# B&R Automation Studio project Panasonic_LinkaPowerCP2_A2021055 (part 22)

#### AtlasCopcoKomunikacia.st
```iecst
ACTION AtlasCopcoKomunikacia:

    M5_PrevodMomentu();
    M4_PrevodMomentu();
    M6_PrevodMomentu();

	//*********************************************************Skrutkovacka M5******************************************************************//
	//Vstupy z AtlasCopco do PLC//
    P2_Srobovanie.Skrutkovacka_M5.Stav_VysledokPotvrdeny:= P2_Srobovanie.PAR.M5_AtlasCopcoInputs[0].0;
    P2_Srobovanie.Skrutkovacka_M5.Stav_EmergencyStop:= P2_Srobovanie.PAR.M5_AtlasCopcoInputs[0].1;
    P2_Srobovanie.Skrutkovacka_M5.Stav_READY_to_START:= P2_Srobovanie.PAR.M5_AtlasCopcoInputs[0].2;
    P2_Srobovanie.Skrutkovacka_M5.Stav_MANUAL:= P2_Srobovanie.PAR.M5_AtlasCopcoInputs[0].3;
    P2_Srobovanie.Skrutkovacka_M5.Stav_UtahovanieUkoncene:= P2_Srobovanie.PAR.M5_AtlasCopcoInputs[0].4;
    P2_Srobovanie.Skrutkovacka_M5.Stav_VysledokUtahovania_NG:= P2_Srobovanie.PAR.M5_AtlasCopcoInputs[0].5;
    P2_Srobovanie.Skrutkovacka_M5.Stav_VysledokUtahovania_OK:= P2_Srobovanie.PAR.M5_AtlasCopcoInputs[0].6;
    P2_Srobovanie.Skrutkovacka_M5.Stav_SmerOtacania_VPRED:= P2_Srobovanie.PAR.M5_AtlasCopcoInputs[0].7;
    P2_Srobovanie.Skrutkovacka_M5.Stav_BUSY:= P2_Srobovanie.PAR.M5_AtlasCopcoInputs[0].8;
    P2_Srobovanie.Skrutkovacka_M5.Stav_ControlerSwitch_ON:= P2_Srobovanie.PAR.M5_AtlasCopcoInputs[0].9;
    P2_Srobovanie.Skrutkovacka_M5.Stav_Station_READY:= P2_Srobovanie.PAR.M5_AtlasCopcoInputs[0].10;
    P2_Srobovanie.Skrutkovacka_M5.Stav_NastrojPripojeny:= P2_Srobovanie.PAR.M5_AtlasCopcoInputs[0].11;
    P2_Srobovanie.Skrutkovacka_M5.Stav_NastrojUtahuje:= P2_Srobovanie.PAR.M5_AtlasCopcoInputs[0].12;

    //Výstupy z PLC do AtlasCopco//
    P2_Srobovanie.PAR.M5_AtlasCopcoOutputs[0].0:= P2_Srobovanie.Skrutkovacka_M5.RESET_Poruchy;
    P2_Srobovanie.PAR.M5_AtlasCopcoOutputs[0].1:= P2_Srobovanie.Skrutkovacka_M5.RESET_Vysledkov;
    P2_Srobovanie.PAR.M5_AtlasCopcoOutputs[0].2:= P2_Srobovanie.Skrutkovacka_M5.START_Skrutkovania;
    P2_Srobovanie.PAR.M5_AtlasCopcoOutputs[0].3:= P2_Srobovanie.Skrutkovacka_M5.START_Utahovania;

    //Dosiahnutý moment//
//    P2_Srobovanie.STAV.M5_DosiahnutyMoment.0:= P2_Srobovanie.PAR.M5_AtlasCopcoInputs[1].24;
//    P2_Srobovanie.STAV.M5_DosiahnutyMoment.1:= P2_Srobovanie.PAR.M5_AtlasCopcoInputs[1].25;
//    P2_Srobovanie.STAV.M5_DosiahnutyMoment.2:= P2_Srobovanie.PAR.M5_AtlasCopcoInputs[1].26;
//    P2_Srobovanie.STAV.M5_DosiahnutyMoment.3:= P2_Srobovanie.PAR.M5_AtlasCopcoInputs[1].27;
//    P2_Srobovanie.STAV.M5_DosiahnutyMoment.4:= P2_Srobovanie.PAR.M5_AtlasCopcoInputs[1].28;
//    P2_Srobovanie.STAV.M5_DosiahnutyMoment.5:= P2_Srobovanie.PAR.M5_AtlasCopcoInputs[1].29;
//    P2_Srobovanie.STAV.M5_DosiahnutyMoment.6:= P2_Srobovanie.PAR.M5_AtlasCopcoInputs[1].30;
//    P2_Srobovanie.STAV.M5_DosiahnutyMoment.7:= P2_Srobovanie.PAR.M5_AtlasCopcoInputs[1].31;
//    P2_Srobovanie.STAV.M5_DosiahnutyMoment.8:= P2_Srobovanie.PAR.M5_AtlasCopcoInputs[1].16;
//    P2_Srobovanie.STAV.M5_DosiahnutyMoment.9:= P2_Srobovanie.PAR.M5_AtlasCopcoInputs[1].17;
//    P2_Srobovanie.STAV.M5_DosiahnutyMoment.10:= P2_Srobovanie.PAR.M5_AtlasCopcoInputs[1].18;
//    P2_Srobovanie.STAV.M5_DosiahnutyMoment.11:= P2_Srobovanie.PAR.M5_AtlasCopcoInputs[1].19;
//    P2_Srobovanie.STAV.M5_DosiahnutyMoment.12:= P2_Srobovanie.PAR.M5_AtlasCopcoInputs[1].20;
//    P2_Srobovanie.STAV.M5_DosiahnutyMoment.13:= P2_Srobovanie.PAR.M5_AtlasCopcoInputs[1].21;
//    P2_Srobovanie.STAV.M5_DosiahnutyMoment.14:= P2_Srobovanie.PAR.M5_AtlasCopcoInputs[1].22;
//    P2_Srobovanie.STAV.M5_DosiahnutyMoment.15:= P2_Srobovanie.PAR.M5_AtlasCopcoInputs[1].23;
//    P2_Srobovanie.STAV.M5_DosiahnutyMoment.16:= P2_Srobovanie.PAR.M5_AtlasCopcoInputs[1].8;
//    P2_Srobovanie.STAV.M5_DosiahnutyMoment.17:= P2_Srobovanie.PAR.M5_AtlasCopcoInputs[1].9;
//    P2_Srobovanie.STAV.M5_DosiahnutyMoment.18:= P2_Srobovanie.PAR.M5_AtlasCopcoInputs[1].10;
//    P2_Srobovanie.STAV.M5_DosiahnutyMoment.19:= P2_Srobovanie.PAR.M5_AtlasCopcoInputs[1].11;
//    P2_Srobovanie.STAV.M5_DosiahnutyMoment.20:= P2_Srobovanie.PAR.M5_AtlasCopcoInputs[1].12;
//    P2_Srobovanie.STAV.M5_DosiahnutyMoment.21:= P2_Srobovanie.PAR.M5_AtlasCopcoInputs[1].13;
//    P2_Srobovanie.STAV.M5_DosiahnutyMoment.22:= P2_Srobovanie.PAR.M5_AtlasCopcoInputs[1].14;
//    P2_Srobovanie.STAV.M5_DosiahnutyMoment.23:= P2_Srobovanie.PAR.M5_AtlasCopcoInputs[1].15;
//    P2_Srobovanie.STAV.M5_DosiahnutyMoment.24:= P2_Srobovanie.PAR.M5_AtlasCopcoInputs[1].0;
//    P2_Srobovanie.STAV.M5_DosiahnutyMoment.25:= P2_Srobovanie.PAR.M5_AtlasCopcoInputs[1].1;
//    P2_Srobovanie.STAV.M5_DosiahnutyMoment.26:= P2_Srobovanie.PAR.M5_AtlasCopcoInputs[1].2;
//    P2_Srobovanie.STAV.M5_DosiahnutyMoment.27:= P2_Srobovanie.PAR.M5_AtlasCopcoInputs[1].3;
//    P2_Srobovanie.STAV.M5_DosiahnutyMoment.28:= P2_Srobovanie.PAR.M5_AtlasCopcoInputs[1].4;
//    P2_Srobovanie.STAV.M5_DosiahnutyMoment.29:= P2_Srobovanie.PAR.M5_AtlasCopcoInputs[1].5;
//    P2_Srobovanie.STAV.M5_DosiahnutyMoment.30:= P2_Srobovanie.PAR.M5_AtlasCopcoInputs[1].6;
//    P2_Srobovanie.STAV.M5_DosiahnutyMoment.31:= P2_Srobovanie.PAR.M5_AtlasCopcoInputs[1].7;
//    M5_DosiahnutyMoment_REAL:= UDINT_TO_REAL(P2_Srobovanie.STAV.M5_DosiahnutyMoment);
//    IF M5_DosiahnutyMoment_REAL > 0 THEN
//        P2_Srobovanie.STAV.M5_DosiahnutyMoment_REAL:= M5_DosiahnutyMoment_REAL/100;
//    ELSE
//        P2_Srobovanie.STAV.M5_DosiahnutyMoment_REAL:= 0.0;
//    END_IF

    M5_PrevodMomentu.AtlasAktualnyMoment:=P2_Srobovanie.PAR.M5_AtlasCopcoInputs[1];
    P2_Srobovanie.STAV.M5_DosiahnutyMoment_REAL:=M5_PrevodMomentu.AktualnyMoment;

    //Moment - Tolerancia MAX//
//    P2_Srobovanie.STAV.M5_Moment_ToleranciaMAX.0:= P2_Srobovanie.PAR.M5_AtlasCopcoInputs[3].24;
//    P2_Srobovanie.STAV.M5_Moment_ToleranciaMAX.1:= P2_Srobovanie.PAR.M5_AtlasCopcoInputs[3].25;
//    P2_Srobovanie.STAV.M5_Moment_ToleranciaMAX.2:= P2_Srobovanie.PAR.M5_AtlasCopcoInputs[3].26;
//    P2_Srobovanie.STAV.M5_Moment_ToleranciaMAX.3:= P2_Srobovanie.PAR.M5_AtlasCopcoInputs[3].27;
//    P2_Srobovanie.STAV.M5_Moment_ToleranciaMAX.4:= P2_Srobovanie.PAR.M5_AtlasCopcoInputs[3].28;
//    P2_Srobovanie.STAV.M5_Moment_ToleranciaMAX.5:= P2_Srobovanie.PAR.M5_AtlasCopcoInputs[3].29;
//    P2_Srobovanie.STAV.M5_Moment_ToleranciaMAX.6:= P2_Srobovanie.PAR.M5_AtlasCopcoInputs[3].30;
//    P2_Srobovanie.STAV.M5_Moment_ToleranciaMAX.7:= P2_Srobovanie.PAR.M5_AtlasCopcoInputs[3].31;
//    P2_Srobovanie.STAV.M5_Moment_ToleranciaMAX.8:= P2_Srobovanie.PAR.M5_AtlasCopcoInputs[3].16;
//    P2_Srobovanie.STAV.M5_Moment_ToleranciaMAX.9:= P2_Srobovanie.PAR.M5_AtlasCopcoInputs[3].17;
//    P2_Srobovanie.STAV.M5_Moment_ToleranciaMAX.10:= P2_Srobovanie.PAR.M5_AtlasCopcoInputs[3].18;
//    P2_Srobovanie.STAV.M5_Moment_ToleranciaMAX.11:= P2_Srobovanie.PAR.M5_AtlasCopcoInputs[3].19;
//    P2_Srobovanie.STAV.M5_Moment_ToleranciaMAX.12:= P2_Srobovanie.PAR.M5_AtlasCopcoInputs[3].20;
//    P2_Srobovanie.STAV.M5_Moment_ToleranciaMAX.13:= P2_Srobovanie.PAR.M5_AtlasCopcoInputs[3].21;
//    P2_Srobovanie.STAV.M5_Moment_ToleranciaMAX.14:= P2_Srobovanie.PAR.M5_AtlasCopcoInputs[3].22;
//    P2_Srobovanie.STAV.M5_Moment_ToleranciaMAX.15:= P2_Srobovanie.PAR.M5_AtlasCopcoInputs[3].23;
//    P2_Srobovanie.STAV.M5_Moment_ToleranciaMAX.16:= P2_Srobovanie.PAR.M5_AtlasCopcoInputs[3].8;
//    P2_Srobovanie.STAV.M5_Moment_ToleranciaMAX.17:= P2_Srobovanie.PAR.M5_AtlasCopcoInputs[3].9;
//    P2_Srobovanie.STAV.M5_Moment_ToleranciaMAX.18:= P2_Srobovanie.PAR.M5_AtlasCopcoInputs[3].10;
//    P2_Srobovanie.STAV.M5_Moment_ToleranciaMAX.19:= P2_Srobovanie.PAR.M5_AtlasCopcoInputs[3].11;
//    P2_Srobovanie.STAV.M5_Moment_ToleranciaMAX.20:= P2_Srobovanie.PAR.M5_AtlasCopcoInputs[3].12;
//    P2_Srobovanie.STAV.M5_Moment_ToleranciaMAX.21:= P2_Srobovanie.PAR.M5_AtlasCopcoInputs[3].13;
//    P2_Srobovanie.STAV.M5_Moment_ToleranciaMAX.22:= P2_Srobovanie.PAR.M5_AtlasCopcoInputs[3].14;
//    P2_Srobovanie.STAV.M5_Moment_ToleranciaMAX.23:= P2_Srobovanie.PAR.M5_AtlasCopcoInputs[3].15;
//    P2_Srobovanie.STAV.M5_Moment_ToleranciaMAX.24:= P2_Srobovanie.PAR.M5_AtlasCopcoInputs[3].0;
//    P2_Srobovanie.STAV.M5_Moment_ToleranciaMAX.25:= P2_Srobovanie.PAR.M5_AtlasCopcoInputs[3].1;
//    P2_Srobovanie.STAV.M5_Moment_ToleranciaMAX.26:= P2_Srobovanie.PAR.M5_AtlasCopcoInputs[3].2;
//    P2_Srobovanie.STAV.M5_Moment_ToleranciaMAX.27:= P2_Srobovanie.PAR.M5_AtlasCopcoInputs[3].3;
//    P2_Srobovanie.STAV.M5_Moment_ToleranciaMAX.28:= P2_Srobovanie.PAR.M5_AtlasCopcoInputs[3].4;
//    P2_Srobovanie.STAV.M5_Moment_ToleranciaMAX.29:= P2_Srobovanie.PAR.M5_AtlasCopcoInputs[3].5;
//    P2_Srobovanie.STAV.M5_Moment_ToleranciaMAX.30:= P2_Srobovanie.PAR.M5_AtlasCopcoInputs[3].6;
//    P2_Srobovanie.STAV.M5_Moment_ToleranciaMAX.31:= P2_Srobovanie.PAR.M5_AtlasCopcoInputs[3].7;
//    M5_Moment_ToleranciaMAX_REAL:= UDINT_TO_REAL(P2_Srobovanie.STAV.M5_Moment_ToleranciaMAX);
//    IF M5_Moment_ToleranciaMAX_REAL > 0 THEN
//        P2_Srobovanie.STAV.M5_Moment_ToleranciaMAX_REAL:= M5_Moment_ToleranciaMAX_REAL/100;
//    ELSE
//        P2_Srobovanie.STAV.M5_Moment_ToleranciaMAX_REAL:= 0.0;
//    END_IF

    M5_PrevodMomentu.AtlasMaximalnaTolerancia:=P2_Srobovanie.PAR.M5_AtlasCopcoInputs[3];
    P2_Srobovanie.STAV.M5_Moment_ToleranciaMAX_REAL:=M5_PrevodMomentu.ToleranciaMAX;

    //Moment - Tolerancia MIN//
//    P2_Srobovanie.STAV.M5_Moment_ToleranciaMIN.0:= P2_Srobovanie.PAR.M5_AtlasCopcoInputs[4].24;
//    P2_Srobovanie.STAV.M5_Moment_ToleranciaMIN.1:= P2_Srobovanie.PAR.M5_AtlasCopcoInputs[4].25;
//    P2_Srobovanie.STAV.M5_Moment_ToleranciaMIN.2:= P2_Srobovanie.PAR.M5_AtlasCopcoInputs[4].26;
//    P2_Srobovanie.STAV.M5_Moment_ToleranciaMIN.3:= P2_Srobovanie.PAR.M5_AtlasCopcoInputs[4].27;
//    P2_Srobovanie.STAV.M5_Moment_ToleranciaMIN.4:= P2_Srobovanie.PAR.M5_AtlasCopcoInputs[4].28;
//    P2_Srobovanie.STAV.M5_Moment_ToleranciaMIN.5:= P2_Srobovanie.PAR.M5_AtlasCopcoInputs[4].29;
//    P2_Srobovanie.STAV.M5_Moment_ToleranciaMIN.6:= P2_Srobovanie.PAR.M5_AtlasCopcoInputs[4].30;
//    P2_Srobovanie.STAV.M5_Moment_ToleranciaMIN.7:= P2_Srobovanie.PAR.M5_AtlasCopcoInputs[4].31;
//    P2_Srobovanie.STAV.M5_Moment_ToleranciaMIN.8:= P2_Srobovanie.PAR.M5_AtlasCopcoInputs[4].16;
//    P2_Srobovanie.STAV.M5_Moment_ToleranciaMIN.9:= P2_Srobovanie.PAR.M5_AtlasCopcoInputs[4].17;
//    P2_Srobovanie.STAV.M5_Moment_ToleranciaMIN.10:= P2_Srobovanie.PAR.M5_AtlasCopcoInputs[4].18;
//    P2_Srobovanie.STAV.M5_Moment_ToleranciaMIN.11:= P2_Srobovanie.PAR.M5_AtlasCopcoInputs[4].19;
//    P2_Srobovanie.STAV.M5_Moment_ToleranciaMIN.12:= P2_Srobovanie.PAR.M5_AtlasCopcoInputs[4].20;
//    P2_Srobovanie.STAV.M5_Moment_ToleranciaMIN.13:= P2_Srobovanie.PAR.M5_AtlasCopcoInputs[4].21;
//    P2_Srobovanie.STAV.M5_Moment_ToleranciaMIN.14:= P2_Srobovanie.PAR.M5_AtlasCopcoInputs[4].22;
//    P2_Srobovanie.STAV.M5_Moment_ToleranciaMIN.15:= P2_Srobovanie.PAR.M5_AtlasCopcoInputs[4].23;
//    P2_Srobovanie.STAV.M5_Moment_ToleranciaMIN.16:= P2_Srobovanie.PAR.M5_AtlasCopcoInputs[4].8;
//    P2_Srobovanie.STAV.M5_Moment_ToleranciaMIN.17:= P2_Srobovanie.PAR.M5_AtlasCopcoInputs[4].9;
//    P2_Srobovanie.STAV.M5_Moment_ToleranciaMIN.18:= P2_Srobovanie.PAR.M5_AtlasCopcoInputs[4].10;
//    P2_Srobovanie.STAV.M5_Moment_ToleranciaMIN.19:= P2_Srobovanie.PAR.M5_AtlasCopcoInputs[4].11;
//    P2_Srobovanie.STAV.M5_Moment_ToleranciaMIN.20:= P2_Srobovanie.PAR.M5_AtlasCopcoInputs[4].12;
//    P2_Srobovanie.STAV.M5_Moment_ToleranciaMIN.21:= P2_Srobovanie.PAR.M5_AtlasCopcoInputs[4].13;
//    P2_Srobovanie.STAV.M5_Moment_ToleranciaMIN.22:= P2_Srobovanie.PAR.M5_AtlasCopcoInputs[4].14;
//    P2_Srobovanie.STAV.M5_Moment_ToleranciaMIN.23:= P2_Srobovanie.PAR.M5_AtlasCopcoInputs[4].15;
//    P2_Srobovanie.STAV.M5_Moment_ToleranciaMIN.24:= P2_Srobovanie.PAR.M5_AtlasCopcoInputs[4].0;
//    P2_Srobovanie.STAV.M5_Moment_ToleranciaMIN.25:= P2_Srobovanie.PAR.M5_AtlasCopcoInputs[4].1;
//    P2_Srobovanie.STAV.M5_Moment_ToleranciaMIN.26:= P2_Srobovanie.PAR.M5_AtlasCopcoInputs[4].2;
//    P2_Srobovanie.STAV.M5_Moment_ToleranciaMIN.27:= P2_Srobovanie.PAR.M5_AtlasCopcoInputs[4].3;
//    P2_Srobovanie.STAV.M5_Moment_ToleranciaMIN.28:= P2_Srobovanie.PAR.M5_AtlasCopcoInputs[4].4;
//    P2_Srobovanie.STAV.M5_Moment_ToleranciaMIN.29:= P2_Srobovanie.PAR.M5_AtlasCopcoInputs[4].5;
//    P2_Srobovanie.STAV.M5_Moment_ToleranciaMIN.30:= P2_Srobovanie.PAR.M5_AtlasCopcoInputs[4].6;
//    P2_Srobovanie.STAV.M5_Moment_ToleranciaMIN.31:= P2_Srobovanie.PAR.M5_AtlasCopcoInputs[4].7;
//    M5_Moment_ToleranciaMIN_REAL:= UDINT_TO_REAL(P2_Srobovanie.STAV.M5_Moment_ToleranciaMIN);
//    IF M5_Moment_ToleranciaMIN_REAL > 0 THEN
//        P2_Srobovanie.STAV.M5_Moment_ToleranciaMIN_REAL:= M5_Moment_ToleranciaMIN_REAL /100;
//    ELSE
//        P2_Srobovanie.STAV.M5_Moment_ToleranciaMIN_REAL:= 0.0;
    //    END_IF

    M5_PrevodMomentu.AtlasMinimalnaTolerancia:=P2_Srobovanie.PAR.M5_AtlasCopcoInputs[4];
    P2_Srobovanie.STAV.M5_Moment_ToleranciaMIN_REAL:=M5_PrevodMomentu.ToleranciaMIN;

    //Dosiahnutý úhol//
    P2_Srobovanie.STAV.M5_DosiahnutyUhol.0:= P2_Srobovanie.PAR.M5_AtlasCopcoInputs[0].24;
    P2_Srobovanie.STAV.M5_DosiahnutyUhol.1:= P2_Srobovanie.PAR.M5_AtlasCopcoInputs[0].25;
    P2_Srobovanie.STAV.M5_DosiahnutyUhol.2:= P2_Srobovanie.PAR.M5_AtlasCopcoInputs[0].26;
    P2_Srobovanie.STAV.M5_DosiahnutyUhol.3:= P2_Srobovanie.PAR.M5_AtlasCopcoInputs[0].27;
    P2_Srobovanie.STAV.M5_DosiahnutyUhol.4:= P2_Srobovanie.PAR.M5_AtlasCopcoInputs[0].28;
    P2_Srobovanie.STAV.M5_DosiahnutyUhol.5:= P2_Srobovanie.PAR.M5_AtlasCopcoInputs[0].29;
    P2_Srobovanie.STAV.M5_DosiahnutyUhol.6:= P2_Srobovanie.PAR.M5_AtlasCopcoInputs[0].30;
    P2_Srobovanie.STAV.M5_DosiahnutyUhol.7:= P2_Srobovanie.PAR.M5_AtlasCopcoInputs[0].31;
    P2_Srobovanie.STAV.M5_DosiahnutyUhol.8:= P2_Srobovanie.PAR.M5_AtlasCopcoInputs[0].16;
    P2_Srobovanie.STAV.M5_DosiahnutyUhol.9:= P2_Srobovanie.PAR.M5_AtlasCopcoInputs[0].17;
    P2_Srobovanie.STAV.M5_DosiahnutyUhol.10:= P2_Srobovanie.PAR.M5_AtlasCopcoInputs[0].18;
    P2_Srobovanie.STAV.M5_DosiahnutyUhol.11:= P2_Srobovanie.PAR.M5_AtlasCopcoInputs[0].19;
    P2_Srobovanie.STAV.M5_DosiahnutyUhol.12:= P2_Srobovanie.PAR.M5_AtlasCopcoInputs[0].20;
    P2_Srobovanie.STAV.M5_DosiahnutyUhol.13:= P2_Srobovanie.PAR.M5_AtlasCopcoInputs[0].21;
    P2_Srobovanie.STAV.M5_DosiahnutyUhol.14:= P2_Srobovanie.PAR.M5_AtlasCopcoInputs[0].22;
    P2_Srobovanie.STAV.M5_DosiahnutyUhol.15:= P2_Srobovanie.PAR.M5_AtlasCopcoInputs[0].23;

    //Uhol - Tolerancia MAX//
    P2_Srobovanie.STAV.M5_Uhol_ToleranciaMAX.0:= P2_Srobovanie.PAR.M5_AtlasCopcoInputs[2].8;
    P2_Srobovanie.STAV.M5_Uhol_ToleranciaMAX.1:= P2_Srobovanie.PAR.M5_AtlasCopcoInputs[2].9;
    P2_Srobovanie.STAV.M5_Uhol_ToleranciaMAX.2:= P2_Srobovanie.PAR.M5_AtlasCopcoInputs[2].10;
    P2_Srobovanie.STAV.M5_Uhol_ToleranciaMAX.3:= P2_Srobovanie.PAR.M5_AtlasCopcoInputs[2].11;
    P2_Srobovanie.STAV.M5_Uhol_ToleranciaMAX.4:= P2_Srobovanie.PAR.M5_AtlasCopcoInputs[2].12;
    P2_Srobovanie.STAV.M5_Uhol_ToleranciaMAX.5:= P2_Srobovanie.PAR.M5_AtlasCopcoInputs[2].13;
    P2_Srobovanie.STAV.M5_Uhol_ToleranciaMAX.6:= P2_Srobovanie.PAR.M5_AtlasCopcoInputs[2].14;
    P2_Srobovanie.STAV.M5_Uhol_ToleranciaMAX.7:= P2_Srobovanie.PAR.M5_AtlasCopcoInputs[2].15;
    P2_Srobovanie.STAV.M5_Uhol_ToleranciaMAX.8:= P2_Srobovanie.PAR.M5_AtlasCopcoInputs[2].0;
    P2_Srobovanie.STAV.M5_Uhol_ToleranciaMAX.9:= P2_Srobovanie.PAR.M5_AtlasCopcoInputs[2].1;
    P2_Srobovanie.STAV.M5_Uhol_ToleranciaMAX.10:= P2_Srobovanie.PAR.M5_AtlasCopcoInputs[2].2;
    P2_Srobovanie.STAV.M5_Uhol_ToleranciaMAX.11:= P2_Srobovanie.PAR.M5_AtlasCopcoInputs[2].3;
    P2_Srobovanie.STAV.M5_Uhol_ToleranciaMAX.12:= P2_Srobovanie.PAR.M5_AtlasCopcoInputs[2].4;
    P2_Srobovanie.STAV.M5_Uhol_ToleranciaMAX.13:= P2_Srobovanie.PAR.M5_AtlasCopcoInputs[2].5;
    P2_Srobovanie.STAV.M5_Uhol_ToleranciaMAX.14:= P2_Srobovanie.PAR.M5_AtlasCopcoInputs[2].6;
    P2_Srobovanie.STAV.M5_Uhol_ToleranciaMAX.15:= P2_Srobovanie.PAR.M5_AtlasCopcoInputs[2].7;

    //Uhol - Tolerancia MIN//
    P2_Srobovanie.STAV.M5_Uhol_ToleranciaMIN.0:= P2_Srobovanie.PAR.M5_AtlasCopcoInputs[2].24;
    P2_Srobovanie.STAV.M5_Uhol_ToleranciaMIN.1:= P2_Srobovanie.PAR.M5_AtlasCopcoInputs[2].25;
    P2_Srobovanie.STAV.M5_Uhol_ToleranciaMIN.2:= P2_Srobovanie.PAR.M5_AtlasCopcoInputs[2].26;
    P2_Srobovanie.STAV.M5_Uhol_ToleranciaMIN.3:= P2_Srobovanie.PAR.M5_AtlasCopcoInputs[2].27;
    P2_Srobovanie.STAV.M5_Uhol_ToleranciaMIN.4:= P2_Srobovanie.PAR.M5_AtlasCopcoInputs[2].28;
    P2_Srobovanie.STAV.M5_Uhol_ToleranciaMIN.5:= P2_Srobovanie.PAR.M5_AtlasCopcoInputs[2].29;
    P2_Srobovanie.STAV.M5_Uhol_ToleranciaMIN.6:= P2_Srobovanie.PAR.M5_AtlasCopcoInputs[2].30;
    P2_Srobovanie.STAV.M5_Uhol_ToleranciaMIN.7:= P2_Srobovanie.PAR.M5_AtlasCopcoInputs[2].31;
    P2_Srobovanie.STAV.M5_Uhol_ToleranciaMIN.8:= P2_Srobovanie.PAR.M5_AtlasCopcoInputs[2].16;
    P2_Srobovanie.STAV.M5_Uhol_ToleranciaMIN.9:= P2_Srobovanie.PAR.M5_AtlasCopcoInputs[2].17;
    P2_Srobovanie.STAV.M5_Uhol_ToleranciaMIN.10:= P2_Srobovanie.PAR.M5_AtlasCopcoInputs[2].18;
    P2_Srobovanie.STAV.M5_Uhol_ToleranciaMIN.11:= P2_Srobovanie.PAR.M5_AtlasCopcoInputs[2].19;
    P2_Srobovanie.STAV.M5_Uhol_ToleranciaMIN.12:= P2_Srobovanie.PAR.M5_AtlasCopcoInputs[2].20;
    P2_Srobovanie.STAV.M5_Uhol_ToleranciaMIN.13:= P2_Srobovanie.PAR.M5_AtlasCopcoInputs[2].21;
    P2_Srobovanie.STAV.M5_Uhol_ToleranciaMIN.14:= P2_Srobovanie.PAR.M5_AtlasCopcoInputs[2].22;
    P2_Srobovanie.STAV.M5_Uhol_ToleranciaMIN.15:= P2_Srobovanie.PAR.M5_AtlasCopcoInputs[2].23;

    //*****************************************************************************Skrutkovacka M4*************************************************************//
    //Vstupy z AtlasCopco do PLC//
    P2_Srobovanie.Skrutkovacka_M4.Stav_VysledokPotvrdeny:= P2_Srobovanie.PAR.M4_AtlasCopcoInputs[0].0;
    P2_Srobovanie.Skrutkovacka_M4.Stav_EmergencyStop:= P2_Srobovanie.PAR.M4_AtlasCopcoInputs[0].1;
    P2_Srobovanie.Skrutkovacka_M4.Stav_READY_to_START:= P2_Srobovanie.PAR.M4_AtlasCopcoInputs[0].2;
    P2_Srobovanie.Skrutkovacka_M4.Stav_MANUAL:= P2_Srobovanie.PAR.M4_AtlasCopcoInputs[0].3;
    P2_Srobovanie.Skrutkovacka_M4.Stav_UtahovanieUkoncene:= P2_Srobovanie.PAR.M4_AtlasCopcoInputs[0].4;
    P2_Srobovanie.Skrutkovacka_M4.Stav_VysledokUtahovania_NG:= P2_Srobovanie.PAR.M4_AtlasCopcoInputs[0].5;
    P2_Srobovanie.Skrutkovacka_M4.Stav_VysledokUtahovania_OK:= P2_Srobovanie.PAR.M4_AtlasCopcoInputs[0].6;
    P2_Srobovanie.Skrutkovacka_M4.Stav_SmerOtacania_VPRED:= P2_Srobovanie.PAR.M4_AtlasCopcoInputs[0].7;
    P2_Srobovanie.Skrutkovacka_M4.Stav_BUSY:= P2_Srobovanie.PAR.M4_AtlasCopcoInputs[0].8;
    P2_Srobovanie.Skrutkovacka_M4.Stav_ControlerSwitch_ON:= P2_Srobovanie.PAR.M4_AtlasCopcoInputs[0].9;
    P2_Srobovanie.Skrutkovacka_M4.Stav_Station_READY:= P2_Srobovanie.PAR.M4_AtlasCopcoInputs[0].10;
    P2_Srobovanie.Skrutkovacka_M4.Stav_NastrojPripojeny:= P2_Srobovanie.PAR.M4_AtlasCopcoInputs[0].11;
    P2_Srobovanie.Skrutkovacka_M4.Stav_NastrojUtahuje:= P2_Srobovanie.PAR.M4_AtlasCopcoInputs[0].12;

    //Výstupy z PLC do AtlasCopco//
    P2_Srobovanie.PAR.M4_AtlasCopcoOutputs[0].0:= P2_Srobovanie.Skrutkovacka_M4.RESET_Poruchy;
    P2_Srobovanie.PAR.M4_AtlasCopcoOutputs[0].1:= P2_Srobovanie.Skrutkovacka_M4.RESET_Vysledkov;
    P2_Srobovanie.PAR.M4_AtlasCopcoOutputs[0].2:= P2_Srobovanie.Skrutkovacka_M4.START_Skrutkovania;
    P2_Srobovanie.PAR.M4_AtlasCopcoOutputs[0].3:= P2_Srobovanie.Skrutkovacka_M4.START_Utahovania;

    //Dosiahnutý moment//
//    P2_Srobovanie.STAV.M4_DosiahnutyMoment.0:= P2_Srobovanie.PAR.M4_AtlasCopcoInputs[1].24;
//    P2_Srobovanie.STAV.M4_DosiahnutyMoment.1:= P2_Srobovanie.PAR.M4_AtlasCopcoInputs[1].25;
//    P2_Srobovanie.STAV.M4_DosiahnutyMoment.2:= P2_Srobovanie.PAR.M4_AtlasCopcoInputs[1].26;
//    P2_Srobovanie.STAV.M4_DosiahnutyMoment.3:= P2_Srobovanie.PAR.M4_AtlasCopcoInputs[1].27;
//    P2_Srobovanie.STAV.M4_DosiahnutyMoment.4:= P2_Srobovanie.PAR.M4_AtlasCopcoInputs[1].28;
//    P2_Srobovanie.STAV.M4_DosiahnutyMoment.5:= P2_Srobovanie.PAR.M4_AtlasCopcoInputs[1].29;
//    P2_Srobovanie.STAV.M4_DosiahnutyMoment.6:= P2_Srobovanie.PAR.M4_AtlasCopcoInputs[1].30;
//    P2_Srobovanie.STAV.M4_DosiahnutyMoment.7:= P2_Srobovanie.PAR.M4_AtlasCopcoInputs[1].31;
//    P2_Srobovanie.STAV.M4_DosiahnutyMoment.8:= P2_Srobovanie.PAR.M4_AtlasCopcoInputs[1].16;
//    P2_Srobovanie.STAV.M4_DosiahnutyMoment.9:= P2_Srobovanie.PAR.M4_AtlasCopcoInputs[1].17;
//    P2_Srobovanie.STAV.M4_DosiahnutyMoment.10:= P2_Srobovanie.PAR.M4_AtlasCopcoInputs[1].18;
//    P2_Srobovanie.STAV.M4_DosiahnutyMoment.11:= P2_Srobovanie.PAR.M4_AtlasCopcoInputs[1].19;
//    P2_Srobovanie.STAV.M4_DosiahnutyMoment.12:= P2_Srobovanie.PAR.M4_AtlasCopcoInputs[1].20;
//    P2_Srobovanie.STAV.M4_DosiahnutyMoment.13:= P2_Srobovanie.PAR.M4_AtlasCopcoInputs[1].21;
//    P2_Srobovanie.STAV.M4_DosiahnutyMoment.14:= P2_Srobovanie.PAR.M4_AtlasCopcoInputs[1].22;
//    P2_Srobovanie.STAV.M4_DosiahnutyMoment.15:= P2_Srobovanie.PAR.M4_AtlasCopcoInputs[1].23;
//    P2_Srobovanie.STAV.M4_DosiahnutyMoment.16:= P2_Srobovanie.PAR.M4_AtlasCopcoInputs[1].8;
//    P2_Srobovanie.STAV.M4_DosiahnutyMoment.17:= P2_Srobovanie.PAR.M4_AtlasCopcoInputs[1].9;
//    P2_Srobovanie.STAV.M4_DosiahnutyMoment.18:= P2_Srobovanie.PAR.M4_AtlasCopcoInputs[1].10;
//    P2_Srobovanie.STAV.M4_DosiahnutyMoment.19:= P2_Srobovanie.PAR.M4_AtlasCopcoInputs[1].11;
//    P2_Srobovanie.STAV.M4_DosiahnutyMoment.20:= P2_Srobovanie.PAR.M4_AtlasCopcoInputs[1].12;
//    P2_Srobovanie.STAV.M4_DosiahnutyMoment.21:= P2_Srobovanie.PAR.M4_AtlasCopcoInputs[1].13;
//    P2_Srobovanie.STAV.M4_DosiahnutyMoment.22:= P2_Srobovanie.PAR.M4_AtlasCopcoInputs[1].14;
//    P2_Srobovanie.STAV.M4_DosiahnutyMoment.23:= P2_Srobovanie.PAR.M4_AtlasCopcoInputs[1].15;
//    P2_Srobovanie.STAV.M4_DosiahnutyMoment.24:= P2_Srobovanie.PAR.M4_AtlasCopcoInputs[1].0;
//    P2_Srobovanie.STAV.M4_DosiahnutyMoment.25:= P2_Srobovanie.PAR.M4_AtlasCopcoInputs[1].1;
//    P2_Srobovanie.STAV.M4_DosiahnutyMoment.26:= P2_Srobovanie.PAR.M4_AtlasCopcoInputs[1].2;
//    P2_Srobovanie.STAV.M4_DosiahnutyMoment.27:= P2_Srobovanie.PAR.M4_AtlasCopcoInputs[1].3;
//    P2_Srobovanie.STAV.M4_DosiahnutyMoment.28:= P2_Srobovanie.PAR.M4_AtlasCopcoInputs[1].4;
//    P2_Srobovanie.STAV.M4_DosiahnutyMoment.29:= P2_Srobovanie.PAR.M4_AtlasCopcoInputs[1].5;
//    P2_Srobovanie.STAV.M4_DosiahnutyMoment.30:= P2_Srobovanie.PAR.M4_AtlasCopcoInputs[1].6;
//    P2_Srobovanie.STAV.M4_DosiahnutyMoment.31:= P2_Srobovanie.PAR.M4_AtlasCopcoInputs[1].7;
//    M4_DosiahnutyMoment_REAL:= UDINT_TO_REAL(P2_Srobovanie.STAV.M4_DosiahnutyMoment);
//    IF M4_DosiahnutyMoment_REAL > 0 THEN
//      P2_Srobovanie.STAV.M4_DosiahnutyMoment_REAL:= (M4_DosiahnutyMoment_REAL*2.1)/131082;
//    ELSE
//        P2_Srobovanie.STAV.M4_DosiahnutyMoment_REAL:= 0.0;
//    END_IF
//    (*P2_Srobovanie.STAV.M4_DosiahnutyMoment_REAL:= M4_DosiahnutyMoment_REAL/100;*)

    M4_PrevodMomentu.AtlasAktualnyMoment:=P2_Srobovanie.PAR.M4_AtlasCopcoInputs[1];
    P2_Srobovanie.STAV.M4_DosiahnutyMoment_REAL:=M4_PrevodMomentu.AktualnyMoment;

    //Moment - Tolerancia MAX//
//    P2_Srobovanie.STAV.M4_Moment_ToleranciaMAX.0:= P2_Srobovanie.PAR.M4_AtlasCopcoInputs[3].24;
//    P2_Srobovanie.STAV.M4_Moment_ToleranciaMAX.1:= P2_Srobovanie.PAR.M4_AtlasCopcoInputs[3].25;
//    P2_Srobovanie.STAV.M4_Moment_ToleranciaMAX.2:= P2_Srobovanie.PAR.M4_AtlasCopcoInputs[3].26;
//    P2_Srobovanie.STAV.M4_Moment_ToleranciaMAX.3:= P2_Srobovanie.PAR.M4_AtlasCopcoInputs[3].27;
//    P2_Srobovanie.STAV.M4_Moment_ToleranciaMAX.4:= P2_Srobovanie.PAR.M4_AtlasCopcoInputs[3].28;
//    P2_Srobovanie.STAV.M4_Moment_ToleranciaMAX.5:= P2_Srobovanie.PAR.M4_AtlasCopcoInputs[3].29;
//    P2_Srobovanie.STAV.M4_Moment_ToleranciaMAX.6:= P2_Srobovanie.PAR.M4_AtlasCopcoInputs[3].30;
//    P2_Srobovanie.STAV.M4_Moment_ToleranciaMAX.7:= P2_Srobovanie.PAR.M4_AtlasCopcoInputs[3].31;
//    P2_Srobovanie.STAV.M4_Moment_ToleranciaMAX.8:= P2_Srobovanie.PAR.M4_AtlasCopcoInputs[3].16;
//    P2_Srobovanie.STAV.M4_Moment_ToleranciaMAX.9:= P2_Srobovanie.PAR.M4_AtlasCopcoInputs[3].17;
//    P2_Srobovanie.STAV.M4_Moment_ToleranciaMAX.10:= P2_Srobovanie.PAR.M4_AtlasCopcoInputs[3].18;
//    P2_Srobovanie.STAV.M4_Moment_ToleranciaMAX.11:= P2_Srobovanie.PAR.M4_AtlasCopcoInputs[3].19;
//    P2_Srobovanie.STAV.M4_Moment_ToleranciaMAX.12:= P2_Srobovanie.PAR.M4_AtlasCopcoInputs[3].20;
//    P2_Srobovanie.STAV.M4_Moment_ToleranciaMAX.13:= P2_Srobovanie.PAR.M4_AtlasCopcoInputs[3].21;
//    P2_Srobovanie.STAV.M4_Moment_ToleranciaMAX.14:= P2_Srobovanie.PAR.M4_AtlasCopcoInputs[3].22;
//    P2_Srobovanie.STAV.M4_Moment_ToleranciaMAX.15:= P2_Srobovanie.PAR.M4_AtlasCopcoInputs[3].23;
//    P2_Srobovanie.STAV.M4_Moment_ToleranciaMAX.16:= P2_Srobovanie.PAR.M4_AtlasCopcoInputs[3].8;
//    P2_Srobovanie.STAV.M4_Moment_ToleranciaMAX.17:= P2_Srobovanie.PAR.M4_AtlasCopcoInputs[3].9;
//    P2_Srobovanie.STAV.M4_Moment_ToleranciaMAX.18:= P2_Srobovanie.PAR.M4_AtlasCopcoInputs[3].10;
//    P2_Srobovanie.STAV.M4_Moment_ToleranciaMAX.19:= P2_Srobovanie.PAR.M4_AtlasCopcoInputs[3].11;
//    P2_Srobovanie.STAV.M4_Moment_ToleranciaMAX.20:= P2_Srobovanie.PAR.M4_AtlasCopcoInputs[3].12;
//    P2_Srobovanie.STAV.M4_Moment_ToleranciaMAX.21:= P2_Srobovanie.PAR.M4_AtlasCopcoInputs[3].13;
//    P2_Srobovanie.STAV.M4_Moment_ToleranciaMAX.22:= P2_Srobovanie.PAR.M4_AtlasCopcoInputs[3].14;
//    P2_Srobovanie.STAV.M4_Moment_ToleranciaMAX.23:= P2_Srobovanie.PAR.M4_AtlasCopcoInputs[3].15;
//    P2_Srobovanie.STAV.M4_Moment_ToleranciaMAX.24:= P2_Srobovanie.PAR.M4_AtlasCopcoInputs[3].0;
//    P2_Srobovanie.STAV.M4_Moment_ToleranciaMAX.25:= P2_Srobovanie.PAR.M4_AtlasCopcoInputs[3].1;
//    P2_Srobovanie.STAV.M4_Moment_ToleranciaMAX.26:= P2_Srobovanie.PAR.M4_AtlasCopcoInputs[3].2;
//    P2_Srobovanie.STAV.M4_Moment_ToleranciaMAX.27:= P2_Srobovanie.PAR.M4_AtlasCopcoInputs[3].3;
//    P2_Srobovanie.STAV.M4_Moment_ToleranciaMAX.28:= P2_Srobovanie.PAR.M4_AtlasCopcoInputs[3].4;
//    P2_Srobovanie.STAV.M4_Moment_ToleranciaMAX.29:= P2_Srobovanie.PAR.M4_AtlasCopcoInputs[3].5;
//    P2_Srobovanie.STAV.M4_Moment_ToleranciaMAX.30:= P2_Srobovanie.PAR.M4_AtlasCopcoInputs[3].6;
//    P2_Srobovanie.STAV.M4_Moment_ToleranciaMAX.31:= P2_Srobovanie.PAR.M4_AtlasCopcoInputs[3].7;
//    M4_Moment_ToleranciaMAX_REAL:= UDINT_TO_REAL(P2_Srobovanie.STAV.M4_Moment_ToleranciaMAX);
//    IF M4_Moment_ToleranciaMAX_REAL > 0 THEN
//        P2_Srobovanie.STAV.M4_Moment_ToleranciaMAX_REAL:= (M4_Moment_ToleranciaMAX_REAL*2.1)/131082;
//    ELSE
//        P2_Srobovanie.STAV.M4_Moment_ToleranciaMAX_REAL:= 0.0;
//    END_IF

    M4_PrevodMomentu.AtlasMaximalnaTolerancia:=P2_Srobovanie.PAR.M4_AtlasCopcoInputs[3];
    P2_Srobovanie.STAV.M4_Moment_ToleranciaMAX_REAL:=M4_PrevodMomentu.ToleranciaMAX;

    (*P2_Srobovanie.STAV.M4_Moment_ToleranciaMAX_REAL:= M4_Moment_ToleranciaMAX_REAL /100;*)

    //Moment - Tolerancia MIN//
//    P2_Srobovanie.STAV.M4_Moment_ToleranciaMIN.0:= P2_Srobovanie.PAR.M4_AtlasCopcoInputs[4].24;
//    P2_Srobovanie.STAV.M4_Moment_ToleranciaMIN.1:= P2_Srobovanie.PAR.M4_AtlasCopcoInputs[4].25;
//    P2_Srobovanie.STAV.M4_Moment_ToleranciaMIN.2:= P2_Srobovanie.PAR.M4_AtlasCopcoInputs[4].26;
//    P2_Srobovanie.STAV.M4_Moment_ToleranciaMIN.3:= P2_Srobovanie.PAR.M4_AtlasCopcoInputs[4].27;
//    P2_Srobovanie.STAV.M4_Moment_ToleranciaMIN.4:= P2_Srobovanie.PAR.M4_AtlasCopcoInputs[4].28;
//    P2_Srobovanie.STAV.M4_Moment_ToleranciaMIN.5:= P2_Srobovanie.PAR.M4_AtlasCopcoInputs[4].29;
//    P2_Srobovanie.STAV.M4_Moment_ToleranciaMIN.6:= P2_Srobovanie.PAR.M4_AtlasCopcoInputs[4].30;
//    P2_Srobovanie.STAV.M4_Moment_ToleranciaMIN.7:= P2_Srobovanie.PAR.M4_AtlasCopcoInputs[4].31;
//    P2_Srobovanie.STAV.M4_Moment_ToleranciaMIN.8:= P2_Srobovanie.PAR.M4_AtlasCopcoInputs[4].16;
//    P2_Srobovanie.STAV.M4_Moment_ToleranciaMIN.9:= P2_Srobovanie.PAR.M4_AtlasCopcoInputs[4].17;
//    P2_Srobovanie.STAV.M4_Moment_ToleranciaMIN.10:= P2_Srobovanie.PAR.M4_AtlasCopcoInputs[4].18;
//    P2_Srobovanie.STAV.M4_Moment_ToleranciaMIN.11:= P2_Srobovanie.PAR.M4_AtlasCopcoInputs[4].19;
//    P2_Srobovanie.STAV.M4_Moment_ToleranciaMIN.12:= P2_Srobovanie.PAR.M4_AtlasCopcoInputs[4].20;
//    P2_Srobovanie.STAV.M4_Moment_ToleranciaMIN.13:= P2_Srobovanie.PAR.M4_AtlasCopcoInputs[4].21;
//    P2_Srobovanie.STAV.M4_Moment_ToleranciaMIN.14:= P2_Srobovanie.PAR.M4_AtlasCopcoInputs[4].22;
//    P2_Srobovanie.STAV.M4_Moment_ToleranciaMIN.15:= P2_Srobovanie.PAR.M4_AtlasCopcoInputs[4].23;
//    P2_Srobovanie.STAV.M4_Moment_ToleranciaMIN.16:= P2_Srobovanie.PAR.M4_AtlasCopcoInputs[4].8;
//    P2_Srobovanie.STAV.M4_Moment_ToleranciaMIN.17:= P2_Srobovanie.PAR.M4_AtlasCopcoInputs[4].9;
//    P2_Srobovanie.STAV.M4_Moment_ToleranciaMIN.18:= P2_Srobovanie.PAR.M4_AtlasCopcoInputs[4].10;
//    P2_Srobovanie.STAV.M4_Moment_ToleranciaMIN.19:= P2_Srobovanie.PAR.M4_AtlasCopcoInputs[4].11;
//    P2_Srobovanie.STAV.M4_Moment_ToleranciaMIN.20:= P2_Srobovanie.PAR.M4_AtlasCopcoInputs[4].12;
//    P2_Srobovanie.STAV.M4_Moment_ToleranciaMIN.21:= P2_Srobovanie.PAR.M4_AtlasCopcoInputs[4].13;
//    P2_Srobovanie.STAV.M4_Moment_ToleranciaMIN.22:= P2_Srobovanie.PAR.M4_AtlasCopcoInputs[4].14;
//    P2_Srobovanie.STAV.M4_Moment_ToleranciaMIN.23:= P2_Srobovanie.PAR.M4_AtlasCopcoInputs[4].15;
//    P2_Srobovanie.STAV.M4_Moment_ToleranciaMIN.24:= P2_Srobovanie.PAR.M4_AtlasCopcoInputs[4].0;
//    P2_Srobovanie.STAV.M4_Moment_ToleranciaMIN.25:= P2_Srobovanie.PAR.M4_AtlasCopcoInputs[4].1;
//    P2_Srobovanie.STAV.M4_Moment_ToleranciaMIN.26:= P2_Srobovanie.PAR.M4_AtlasCopcoInputs[4].2;
//    P2_Srobovanie.STAV.M4_Moment_ToleranciaMIN.27:= P2_Srobovanie.PAR.M4_AtlasCopcoInputs[4].3;
//    P2_Srobovanie.STAV.M4_Moment_ToleranciaMIN.28:= P2_Srobovanie.PAR.M4_AtlasCopcoInputs[4].4;
//    P2_Srobovanie.STAV.M4_Moment_ToleranciaMIN.29:= P2_Srobovanie.PAR.M4_AtlasCopcoInputs[4].5;
//    P2_Srobovanie.STAV.M4_Moment_ToleranciaMIN.30:= P2_Srobovanie.PAR.M4_AtlasCopcoInputs[4].6;
//    P2_Srobovanie.STAV.M4_Moment_ToleranciaMIN.31:= P2_Srobovanie.PAR.M4_AtlasCopcoInputs[4].7;
//    M4_Moment_ToleranciaMIN_REAL:= UDINT_TO_REAL(P2_Srobovanie.STAV.M4_Moment_ToleranciaMIN);
//    IF M4_Moment_ToleranciaMIN_REAL > 0 THEN
//        P2_Srobovanie.STAV.M4_Moment_ToleranciaMIN_REAL:= (M4_Moment_ToleranciaMIN_REAL*2.1)/131082;
//    ELSE
//        P2_Srobovanie.STAV.M4_Moment_ToleranciaMIN_REAL:= 0.0;
//    END_IF
//

    M4_PrevodMomentu.AtlasMinimalnaTolerancia:=P2_Srobovanie.PAR.M4_AtlasCopcoInputs[4];
    P2_Srobovanie.STAV.M4_Moment_ToleranciaMIN_REAL:=M4_PrevodMomentu.ToleranciaMIN;

    (*P2_Srobovanie.STAV.M4_Moment_ToleranciaMIN_REAL:= M4_Moment_ToleranciaMIN_REAL /100;*)

    //Dosiahnutý úhol//
    P2_Srobovanie.STAV.M4_DosiahnutyUhol.0:= P2_Srobovanie.PAR.M4_AtlasCopcoInputs[0].24;
    P2_Srobovanie.STAV.M4_DosiahnutyUhol.1:= P2_Srobovanie.PAR.M4_AtlasCopcoInputs[0].25;
    P2_Srobovanie.STAV.M4_DosiahnutyUhol.2:= P2_Srobovanie.PAR.M4_AtlasCopcoInputs[0].26;
    P2_Srobovanie.STAV.M4_DosiahnutyUhol.3:= P2_Srobovanie.PAR.M4_AtlasCopcoInputs[0].27;
    P2_Srobovanie.STAV.M4_DosiahnutyUhol.4:= P2_Srobovanie.PAR.M4_AtlasCopcoInputs[0].28;
    P2_Srobovanie.STAV.M4_DosiahnutyUhol.5:= P2_Srobovanie.PAR.M4_AtlasCopcoInputs[0].29;
    P2_Srobovanie.STAV.M4_DosiahnutyUhol.6:= P2_Srobovanie.PAR.M4_AtlasCopcoInputs[0].30;
    P2_Srobovanie.STAV.M4_DosiahnutyUhol.7:= P2_Srobovanie.PAR.M4_AtlasCopcoInputs[0].31;
    P2_Srobovanie.STAV.M4_DosiahnutyUhol.8:= P2_Srobovanie.PAR.M4_AtlasCopcoInputs[0].16;
    P2_Srobovanie.STAV.M4_DosiahnutyUhol.9:= P2_Srobovanie.PAR.M4_AtlasCopcoInputs[0].17;
    P2_Srobovanie.STAV.M4_DosiahnutyUhol.10:= P2_Srobovanie.PAR.M4_AtlasCopcoInputs[0].18;
    P2_Srobovanie.STAV.M4_DosiahnutyUhol.11:= P2_Srobovanie.PAR.M4_AtlasCopcoInputs[0].19;
    P2_Srobovanie.STAV.M4_DosiahnutyUhol.12:= P2_Srobovanie.PAR.M4_AtlasCopcoInputs[0].20;
    P2_Srobovanie.STAV.M4_DosiahnutyUhol.13:= P2_Srobovanie.PAR.M4_AtlasCopcoInputs[0].21;
    P2_Srobovanie.STAV.M4_DosiahnutyUhol.14:= P2_Srobovanie.PAR.M4_AtlasCopcoInputs[0].22;
    P2_Srobovanie.STAV.M4_DosiahnutyUhol.15:= P2_Srobovanie.PAR.M4_AtlasCopcoInputs[0].23;

    //Uhol - Tolerancia MAX//
    P2_Srobovanie.STAV.M4_Uhol_ToleranciaMAX.0:= P2_Srobovanie.PAR.M4_AtlasCopcoInputs[2].8;
    P2_Srobovanie.STAV.M4_Uhol_ToleranciaMAX.1:= P2_Srobovanie.PAR.M4_AtlasCopcoInputs[2].9;
    P2_Srobovanie.STAV.M4_Uhol_ToleranciaMAX.2:= P2_Srobovanie.PAR.M4_AtlasCopcoInputs[2].10;
    P2_Srobovanie.STAV.M4_Uhol_ToleranciaMAX.3:= P2_Srobovanie.PAR.M4_AtlasCopcoInputs[2].11;
    P2_Srobovanie.STAV.M4_Uhol_ToleranciaMAX.4:= P2_Srobovanie.PAR.M4_AtlasCopcoInputs[2].12;
    P2_Srobovanie.STAV.M4_Uhol_ToleranciaMAX.5:= P2_Srobovanie.PAR.M4_AtlasCopcoInputs[2].13;
    P2_Srobovanie.STAV.M4_Uhol_ToleranciaMAX.6:= P2_Srobovanie.PAR.M4_AtlasCopcoInputs[2].14;
    P2_Srobovanie.STAV.M4_Uhol_ToleranciaMAX.7:= P2_Srobovanie.PAR.M4_AtlasCopcoInputs[2].15;
    P2_Srobovanie.STAV.M4_Uhol_ToleranciaMAX.8:= P2_Srobovanie.PAR.M4_AtlasCopcoInputs[2].0;
    P2_Srobovanie.STAV.M4_Uhol_ToleranciaMAX.9:= P2_Srobovanie.PAR.M4_AtlasCopcoInputs[2].1;
    P2_Srobovanie.STAV.M4_Uhol_ToleranciaMAX.10:= P2_Srobovanie.PAR.M4_AtlasCopcoInputs[2].2;
    P2_Srobovanie.STAV.M4_Uhol_ToleranciaMAX.11:= P2_Srobovanie.PAR.M4_AtlasCopcoInputs[2].3;
    P2_Srobovanie.STAV.M4_Uhol_ToleranciaMAX.12:= P2_Srobovanie.PAR.M4_AtlasCopcoInputs[2].4;
    P2_Srobovanie.STAV.M4_Uhol_ToleranciaMAX.13:= P2_Srobovanie.PAR.M4_AtlasCopcoInputs[2].5;
    P2_Srobovanie.STAV.M4_Uhol_ToleranciaMAX.14:= P2_Srobovanie.PAR.M4_AtlasCopcoInputs[2].6;
    P2_Srobovanie.STAV.M4_Uhol_ToleranciaMAX.15:= P2_Srobovanie.PAR.M4_AtlasCopcoInputs[2].7;

    //Uhol - Tolerancia MIN//
    P2_Srobovanie.STAV.M4_Uhol_ToleranciaMIN.0:= P2_Srobovanie.PAR.M4_AtlasCopcoInputs[2].24;
    P2_Srobovanie.STAV.M4_Uhol_ToleranciaMIN.1:= P2_Srobovanie.PAR.M4_AtlasCopcoInputs[2].25;
    P2_Srobovanie.STAV.M4_Uhol_ToleranciaMIN.2:= P2_Srobovanie.PAR.M4_AtlasCopcoInputs[2].26;
    P2_Srobovanie.STAV.M4_Uhol_ToleranciaMIN.3:= P2_Srobovanie.PAR.M4_AtlasCopcoInputs[2].27;
    P2_Srobovanie.STAV.M4_Uhol_ToleranciaMIN.4:= P2_Srobovanie.PAR.M4_AtlasCopcoInputs[2].28;
    P2_Srobovanie.STAV.M4_Uhol_ToleranciaMIN.5:= P2_Srobovanie.PAR.M4_AtlasCopcoInputs[2].29;
    P2_Srobovanie.STAV.M4_Uhol_ToleranciaMIN.6:= P2_Srobovanie.PAR.M4_AtlasCopcoInputs[2].30;
    P2_Srobovanie.STAV.M4_Uhol_ToleranciaMIN.7:= P2_Srobovanie.PAR.M4_AtlasCopcoInputs[2].31;
    P2_Srobovanie.STAV.M4_Uhol_ToleranciaMIN.8:= P2_Srobovanie.PAR.M4_AtlasCopcoInputs[2].16;
    P2_Srobovanie.STAV.M4_Uhol_ToleranciaMIN.9:= P2_Srobovanie.PAR.M4_AtlasCopcoInputs[2].17;
    P2_Srobovanie.STAV.M4_Uhol_ToleranciaMIN.10:= P2_Srobovanie.PAR.M4_AtlasCopcoInputs[2].18;
    P2_Srobovanie.STAV.M4_Uhol_ToleranciaMIN.11:= P2_Srobovanie.PAR.M4_AtlasCopcoInputs[2].19;
    P2_Srobovanie.STAV.M4_Uhol_ToleranciaMIN.12:= P2_Srobovanie.PAR.M4_AtlasCopcoInputs[2].20;
    P2_Srobovanie.STAV.M4_Uhol_ToleranciaMIN.13:= P2_Srobovanie.PAR.M4_AtlasCopcoInputs[2].21;
    P2_Srobovanie.STAV.M4_Uhol_ToleranciaMIN.14:= P2_Srobovanie.PAR.M4_AtlasCopcoInputs[2].22;
    P2_Srobovanie.STAV.M4_Uhol_ToleranciaMIN.15:= P2_Srobovanie.PAR.M4_AtlasCopcoInputs[2].23;

    //*************************************************************Skrutkovacka M6*******************************************************************************//
    //Vstupy z AtlasCopco do PLC//
    P2_Srobovanie.Skrutkovacka_M6.Stav_VysledokPotvrdeny:= P2_Srobovanie.PAR.M6_AtlasCopcoInputs[0].0;
    P2_Srobovanie.Skrutkovacka_M6.Stav_EmergencyStop:= P2_Srobovanie.PAR.M6_AtlasCopcoInputs[0].1;
    P2_Srobovanie.Skrutkovacka_M6.Stav_READY_to_START:= P2_Srobovanie.PAR.M6_AtlasCopcoInputs[0].2;
    P2_Srobovanie.Skrutkovacka_M6.Stav_MANUAL:= P2_Srobovanie.PAR.M6_AtlasCopcoInputs[0].3;
    P2_Srobovanie.Skrutkovacka_M6.Stav_UtahovanieUkoncene:= P2_Srobovanie.PAR.M6_AtlasCopcoInputs[0].4;
    P2_Srobovanie.Skrutkovacka_M6.Stav_VysledokUtahovania_NG:= P2_Srobovanie.PAR.M6_AtlasCopcoInputs[0].5;
    P2_Srobovanie.Skrutkovacka_M6.Stav_VysledokUtahovania_OK:= P2_Srobovanie.PAR.M6_AtlasCopcoInputs[0].6;
    P2_Srobovanie.Skrutkovacka_M6.Stav_SmerOtacania_VPRED:= P2_Srobovanie.PAR.M6_AtlasCopcoInputs[0].7;
    P2_Srobovanie.Skrutkovacka_M6.Stav_BUSY:= P2_Srobovanie.PAR.M6_AtlasCopcoInputs[0].8;
    P2_Srobovanie.Skrutkovacka_M6.Stav_ControlerSwitch_ON:= P2_Srobovanie.PAR.M6_AtlasCopcoInputs[0].9;
    P2_Srobovanie.Skrutkovacka_M6.Stav_Station_READY:= P2_Srobovanie.PAR.M6_AtlasCopcoInputs[0].10;
    P2_Srobovanie.Skrutkovacka_M6.Stav_NastrojPripojeny:= P2_Srobovanie.PAR.M6_AtlasCopcoInputs[0].11;
    P2_Srobovanie.Skrutkovacka_M6.Stav_NastrojUtahuje:= P2_Srobovanie.PAR.M6_AtlasCopcoInputs[0].12;

    //Výstupy z PLC do AtlasCopco//
    P2_Srobovanie.PAR.M6_AtlasCopcoOutputs[0].0:= P2_Srobovanie.Skrutkovacka_M6.RESET_Poruchy;
    P2_Srobovanie.PAR.M6_AtlasCopcoOutputs[0].1:= P2_Srobovanie.Skrutkovacka_M6.RESET_Vysledkov;
    P2_Srobovanie.PAR.M6_AtlasCopcoOutputs[0].2:= P2_Srobovanie.Skrutkovacka_M6.START_Skrutkovania;
    P2_Srobovanie.PAR.M6_AtlasCopcoOutputs[0].3:= P2_Srobovanie.Skrutkovacka_M6.START_Utahovania;

    //Dosiahnutý moment//
//    P2_Srobovanie.STAV.M6_DosiahnutyMoment.0:= P2_Srobovanie.PAR.M6_AtlasCopcoInputs[1].24;
//    P2_Srobovanie.STAV.M6_DosiahnutyMoment.1:= P2_Srobovanie.PAR.M6_AtlasCopcoInputs[1].25;
//    P2_Srobovanie.STAV.M6_DosiahnutyMoment.2:= P2_Srobovanie.PAR.M6_AtlasCopcoInputs[1].26;
//    P2_Srobovanie.STAV.M6_DosiahnutyMoment.3:= P2_Srobovanie.PAR.M6_AtlasCopcoInputs[1].27;
//    P2_Srobovanie.STAV.M6_DosiahnutyMoment.4:= P2_Srobovanie.PAR.M6_AtlasCopcoInputs[1].28;
//    P2_Srobovanie.STAV.M6_DosiahnutyMoment.5:= P2_Srobovanie.PAR.M6_AtlasCopcoInputs[1].29;
//    P2_Srobovanie.STAV.M6_DosiahnutyMoment.6:= P2_Srobovanie.PAR.M6_AtlasCopcoInputs[1].30;
//    P2_Srobovanie.STAV.M6_DosiahnutyMoment.7:= P2_Srobovanie.PAR.M6_AtlasCopcoInputs[1].31;
//    P2_Srobovanie.STAV.M6_DosiahnutyMoment.8:= P2_Srobovanie.PAR.M6_AtlasCopcoInputs[1].16;
//    P2_Srobovanie.STAV.M6_DosiahnutyMoment.9:= P2_Srobovanie.PAR.M6_AtlasCopcoInputs[1].17;
//    P2_Srobovanie.STAV.M6_DosiahnutyMoment.10:= P2_Srobovanie.PAR.M6_AtlasCopcoInputs[1].18;
//    P2_Srobovanie.STAV.M6_DosiahnutyMoment.11:= P2_Srobovanie.PAR.M6_AtlasCopcoInputs[1].19;
//    P2_Srobovanie.STAV.M6_DosiahnutyMoment.12:= P2_Srobovanie.PAR.M6_AtlasCopcoInputs[1].20;
//    P2_Srobovanie.STAV.M6_DosiahnutyMoment.13:= P2_Srobovanie.PAR.M6_AtlasCopcoInputs[1].21;
//    P2_Srobovanie.STAV.M6_DosiahnutyMoment.14:= P2_Srobovanie.PAR.M6_AtlasCopcoInputs[1].22;
//    P2_Srobovanie.STAV.M6_DosiahnutyMoment.15:= P2_Srobovanie.PAR.M6_AtlasCopcoInputs[1].23;
//    P2_Srobovanie.STAV.M6_DosiahnutyMoment.16:= P2_Srobovanie.PAR.M6_AtlasCopcoInputs[1].8;
//    P2_Srobovanie.STAV.M6_DosiahnutyMoment.17:= P2_Srobovanie.PAR.M6_AtlasCopcoInputs[1].9;
//    P2_Srobovanie.STAV.M6_DosiahnutyMoment.18:= P2_Srobovanie.PAR.M6_AtlasCopcoInputs[1].10;
//    P2_Srobovanie.STAV.M6_DosiahnutyMoment.19:= P2_Srobovanie.PAR.M6_AtlasCopcoInputs[1].11;
//    P2_Srobovanie.STAV.M6_DosiahnutyMoment.20:= P2_Srobovanie.PAR.M6_AtlasCopcoInputs[1].12;
//    P2_Srobovanie.STAV.M6_DosiahnutyMoment.21:= P2_Srobovanie.PAR.M6_AtlasCopcoInputs[1].13;
//    P2_Srobovanie.STAV.M6_DosiahnutyMoment.22:= P2_Srobovanie.PAR.M6_AtlasCopcoInputs[1].14;
//    P2_Srobovanie.STAV.M6_DosiahnutyMoment.23:= P2_Srobovanie.PAR.M6_AtlasCopcoInputs[1].15;
//    P2_Srobovanie.STAV.M6_DosiahnutyMoment.24:= P2_Srobovanie.PAR.M6_AtlasCopcoInputs[1].0;
//    P2_Srobovanie.STAV.M6_DosiahnutyMoment.25:= P2_Srobovanie.PAR.M6_AtlasCopcoInputs[1].1;
//    P2_Srobovanie.STAV.M6_DosiahnutyMoment.26:= P2_Srobovanie.PAR.M6_AtlasCopcoInputs[1].2;
//    P2_Srobovanie.STAV.M6_DosiahnutyMoment.27:= P2_Srobovanie.PAR.M6_AtlasCopcoInputs[1].3;
//    P2_Srobovanie.STAV.M6_DosiahnutyMoment.28:= P2_Srobovanie.PAR.M6_AtlasCopcoInputs[1].4;
//    P2_Srobovanie.STAV.M6_DosiahnutyMoment.29:= P2_Srobovanie.PAR.M6_AtlasCopcoInputs[1].5;
//    P2_Srobovanie.STAV.M6_DosiahnutyMoment.30:= P2_Srobovanie.PAR.M6_AtlasCopcoInputs[1].6;
//    P2_Srobovanie.STAV.M6_DosiahnutyMoment.31:= P2_Srobovanie.PAR.M6_AtlasCopcoInputs[1].7;
//    M6_DosiahnutyMoment_REAL:= UDINT_TO_REAL(P2_Srobovanie.STAV.M6_DosiahnutyMoment);
//    IF M6_DosiahnutyMoment_REAL > 0 THEN
//       P2_Srobovanie.STAV.M6_DosiahnutyMoment_REAL:= (M6_DosiahnutyMoment_REAL*7.2)/458772;
//    ELSE
//        P2_Srobovanie.STAV.M6_DosiahnutyMoment_REAL:= 0.0;
//    END_IF

    M6_PrevodMomentu.AtlasAktualnyMoment:=P2_Srobovanie.PAR.M6_AtlasCopcoInputs[1];
    P2_Srobovanie.STAV.M6_DosiahnutyMoment_REAL:=M6_PrevodMomentu.AktualnyMoment;

    (*P2_Srobovanie.STAV.M6_DosiahnutyMoment_REAL:= M6_DosiahnutyMoment_REAL /100;*)

    //Moment - Tolerancia MAX//
//    P2_Srobovanie.STAV.M6_Moment_ToleranciaMAX.0:= P2_Srobovanie.PAR.M6_AtlasCopcoInputs[3].24;
//    P2_Srobovanie.STAV.M6_Moment_ToleranciaMAX.1:= P2_Srobovanie.PAR.M6_AtlasCopcoInputs[3].25;
//    P2_Srobovanie.STAV.M6_Moment_ToleranciaMAX.2:= P2_Srobovanie.PAR.M6_AtlasCopcoInputs[3].26;
//    P2_Srobovanie.STAV.M6_Moment_ToleranciaMAX.3:= P2_Srobovanie.PAR.M6_AtlasCopcoInputs[3].27;
//    P2_Srobovanie.STAV.M6_Moment_ToleranciaMAX.4:= P2_Srobovanie.PAR.M6_AtlasCopcoInputs[3].28;
//    P2_Srobovanie.STAV.M6_Moment_ToleranciaMAX.5:= P2_Srobovanie.PAR.M6_AtlasCopcoInputs[3].29;
//    P2_Srobovanie.STAV.M6_Moment_ToleranciaMAX.6:= P2_Srobovanie.PAR.M6_AtlasCopcoInputs[3].30;
//    P2_Srobovanie.STAV.M6_Moment_ToleranciaMAX.7:= P2_Srobovanie.PAR.M6_AtlasCopcoInputs[3].31;
//    P2_Srobovanie.STAV.M6_Moment_ToleranciaMAX.8:= P2_Srobovanie.PAR.M6_AtlasCopcoInputs[3].16;
//    P2_Srobovanie.STAV.M6_Moment_ToleranciaMAX.9:= P2_Srobovanie.PAR.M6_AtlasCopcoInputs[3].17;
//    P2_Srobovanie.STAV.M6_Moment_ToleranciaMAX.10:= P2_Srobovanie.PAR.M6_AtlasCopcoInputs[3].18;
//    P2_Srobovanie.STAV.M6_Moment_ToleranciaMAX.11:= P2_Srobovanie.PAR.M6_AtlasCopcoInputs[3].19;
//    P2_Srobovanie.STAV.M6_Moment_ToleranciaMAX.12:= P2_Srobovanie.PAR.M6_AtlasCopcoInputs[3].20;
//    P2_Srobovanie.STAV.M6_Moment_ToleranciaMAX.13:= P2_Srobovanie.PAR.M6_AtlasCopcoInputs[3].21;
//    P2_Srobovanie.STAV.M6_Moment_ToleranciaMAX.14:= P2_Srobovanie.PAR.M6_AtlasCopcoInputs[3].22;
//    P2_Srobovanie.STAV.M6_Moment_ToleranciaMAX.15:= P2_Srobovanie.PAR.M6_AtlasCopcoInputs[3].23;
//    P2_Srobovanie.STAV.M6_Moment_ToleranciaMAX.16:= P2_Srobovanie.PAR.M6_AtlasCopcoInputs[3].8;
//    P2_Srobovanie.STAV.M6_Moment_ToleranciaMAX.17:= P2_Srobovanie.PAR.M6_AtlasCopcoInputs[3].9;
//    P2_Srobovanie.STAV.M6_Moment_ToleranciaMAX.18:= P2_Srobovanie.PAR.M6_AtlasCopcoInputs[3].10;
//    P2_Srobovanie.STAV.M6_Moment_ToleranciaMAX.19:= P2_Srobovanie.PAR.M6_AtlasCopcoInputs[3].11;
//    P2_Srobovanie.STAV.M6_Moment_ToleranciaMAX.20:= P2_Srobovanie.PAR.M6_AtlasCopcoInputs[3].12;
//    P2_Srobovanie.STAV.M6_Moment_ToleranciaMAX.21:= P2_Srobovanie.PAR.M6_AtlasCopcoInputs[3].13;
//    P2_Srobovanie.STAV.M6_Moment_ToleranciaMAX.22:= P2_Srobovanie.PAR.M6_AtlasCopcoInputs[3].14;
//    P2_Srobovanie.STAV.M6_Moment_ToleranciaMAX.23:= P2_Srobovanie.PAR.M6_AtlasCopcoInputs[3].15;
//    P2_Srobovanie.STAV.M6_Moment_ToleranciaMAX.24:= P2_Srobovanie.PAR.M6_AtlasCopcoInputs[3].0;
//    P2_Srobovanie.STAV.M6_Moment_ToleranciaMAX.25:= P2_Srobovanie.PAR.M6_AtlasCopcoInputs[3].1;
//    P2_Srobovanie.STAV.M6_Moment_ToleranciaMAX.26:= P2_Srobovanie.PAR.M6_AtlasCopcoInputs[3].2;
//    P2_Srobovanie.STAV.M6_Moment_ToleranciaMAX.27:= P2_Srobovanie.PAR.M6_AtlasCopcoInputs[3].3;
//    P2_Srobovanie.STAV.M6_Moment_ToleranciaMAX.28:= P2_Srobovanie.PAR.M6_AtlasCopcoInputs[3].4;
//    P2_Srobovanie.STAV.M6_Moment_ToleranciaMAX.29:= P2_Srobovanie.PAR.M6_AtlasCopcoInputs[3].5;
//    P2_Srobovanie.STAV.M6_Moment_ToleranciaMAX.30:= P2_Srobovanie.PAR.M6_AtlasCopcoInputs[3].6;
//    P2_Srobovanie.STAV.M6_Moment_ToleranciaMAX.31:= P2_Srobovanie.PAR.M6_AtlasCopcoInputs[3].7;
//    M6_Moment_ToleranciaMAX_REAL:= UDINT_TO_REAL(P2_Srobovanie.STAV.M6_Moment_ToleranciaMAX);
//    IF M6_Moment_ToleranciaMAX_REAL > 0 THEN
//        P2_Srobovanie.STAV.M6_Moment_ToleranciaMAX_REAL:= (M6_Moment_ToleranciaMAX_REAL*7.2)/458772;
//    ELSE
//        P2_Srobovanie.STAV.M6_Moment_ToleranciaMAX_REAL:= 0.0;
//    END_IF
//

    M6_PrevodMomentu.AtlasMaximalnaTolerancia:=P2_Srobovanie.PAR.M6_AtlasCopcoInputs[3];
    P2_Srobovanie.STAV.M6_Moment_ToleranciaMAX_REAL:=M6_PrevodMomentu.ToleranciaMAX;

    (*P2_Srobovanie.STAV.M6_Moment_ToleranciaMAX_REAL:= M6_Moment_ToleranciaMAX_REAL /100;*)

    //Moment - Tolerancia MIN//
//    P2_Srobovanie.STAV.M6_Moment_ToleranciaMIN.0:= P2_Srobovanie.PAR.M6_AtlasCopcoInputs[4].24;
//    P2_Srobovanie.STAV.M6_Moment_ToleranciaMIN.1:= P2_Srobovanie.PAR.M6_AtlasCopcoInputs[4].25;
//    P2_Srobovanie.STAV.M6_Moment_ToleranciaMIN.2:= P2_Srobovanie.PAR.M6_AtlasCopcoInputs[4].26;
//    P2_Srobovanie.STAV.M6_Moment_ToleranciaMIN.3:= P2_Srobovanie.PAR.M6_AtlasCopcoInputs[4].27;
//    P2_Srobovanie.STAV.M6_Moment_ToleranciaMIN.4:= P2_Srobovanie.PAR.M6_AtlasCopcoInputs[4].28;
//    P2_Srobovanie.STAV.M6_Moment_ToleranciaMIN.5:= P2_Srobovanie.PAR.M6_AtlasCopcoInputs[4].29;
//    P2_Srobovanie.STAV.M6_Moment_ToleranciaMIN.6:= P2_Srobovanie.PAR.M6_AtlasCopcoInputs[4].30;
//    P2_Srobovanie.STAV.M6_Moment_ToleranciaMIN.7:= P2_Srobovanie.PAR.M6_AtlasCopcoInputs[4].31;
//    P2_Srobovanie.STAV.M6_Moment_ToleranciaMIN.8:= P2_Srobovanie.PAR.M6_AtlasCopcoInputs[4].16;
//    P2_Srobovanie.STAV.M6_Moment_ToleranciaMIN.9:= P2_Srobovanie.PAR.M6_AtlasCopcoInputs[4].17;
//    P2_Srobovanie.STAV.M6_Moment_ToleranciaMIN.10:= P2_Srobovanie.PAR.M6_AtlasCopcoInputs[4].18;
//    P2_Srobovanie.STAV.M6_Moment_ToleranciaMIN.11:= P2_Srobovanie.PAR.M6_AtlasCopcoInputs[4].19;
//    P2_Srobovanie.STAV.M6_Moment_ToleranciaMIN.12:= P2_Srobovanie.PAR.M6_AtlasCopcoInputs[4].20;
//    P2_Srobovanie.STAV.M6_Moment_ToleranciaMIN.13:= P2_Srobovanie.PAR.M6_AtlasCopcoInputs[4].21;
//    P2_Srobovanie.STAV.M6_Moment_ToleranciaMIN.14:= P2_Srobovanie.PAR.M6_AtlasCopcoInputs[4].22;
//    P2_Srobovanie.STAV.M6_Moment_ToleranciaMIN.15:= P2_Srobovanie.PAR.M6_AtlasCopcoInputs[4].23;
//    P2_Srobovanie.STAV.M6_Moment_ToleranciaMIN.16:= P2_Srobovanie.PAR.M6_AtlasCopcoInputs[4].8;
//    P2_Srobovanie.STAV.M6_Moment_ToleranciaMIN.17:= P2_Srobovanie.PAR.M6_AtlasCopcoInputs[4].9;
//    P2_Srobovanie.STAV.M6_Moment_ToleranciaMIN.18:= P2_Srobovanie.PAR.M6_AtlasCopcoInputs[4].10;
//    P2_Srobovanie.STAV.M6_Moment_ToleranciaMIN.19:= P2_Srobovanie.PAR.M6_AtlasCopcoInputs[4].11;
//    P2_Srobovanie.STAV.M6_Moment_ToleranciaMIN.20:= P2_Srobovanie.PAR.M6_AtlasCopcoInputs[4].12;
//    P2_Srobovanie.STAV.M6_Moment_ToleranciaMIN.21:= P2_Srobovanie.PAR.M6_AtlasCopcoInputs[4].13;
//    P2_Srobovanie.STAV.M6_Moment_ToleranciaMIN.22:= P2_Srobovanie.PAR.M6_AtlasCopcoInputs[4].14;
//    P2_Srobovanie.STAV.M6_Moment_ToleranciaMIN.23:= P2_Srobovanie.PAR.M6_AtlasCopcoInputs[4].15;
//    P2_Srobovanie.STAV.M6_Moment_ToleranciaMIN.24:= P2_Srobovanie.PAR.M6_AtlasCopcoInputs[4].0;
//    P2_Srobovanie.STAV.M6_Moment_ToleranciaMIN.25:= P2_Srobovanie.PAR.M6_AtlasCopcoInputs[4].1;
//    P2_Srobovanie.STAV.M6_Moment_ToleranciaMIN.26:= P2_Srobovanie.PAR.M6_AtlasCopcoInputs[4].2;
//    P2_Srobovanie.STAV.M6_Moment_ToleranciaMIN.27:= P2_Srobovanie.PAR.M6_AtlasCopcoInputs[4].3;
//    P2_Srobovanie.STAV.M6_Moment_ToleranciaMIN.28:= P2_Srobovanie.PAR.M6_AtlasCopcoInputs[4].4;
//    P2_Srobovanie.STAV.M6_Moment_ToleranciaMIN.29:= P2_Srobovanie.PAR.M6_AtlasCopcoInputs[4].5;
//    P2_Srobovanie.STAV.M6_Moment_ToleranciaMIN.30:= P2_Srobovanie.PAR.M6_AtlasCopcoInputs[4].6;
//    P2_Srobovanie.STAV.M6_Moment_ToleranciaMIN.31:= P2_Srobovanie.PAR.M6_AtlasCopcoInputs[4].7;
//    M6_Moment_ToleranciaMIN_REAL:= UDINT_TO_REAL(P2_Srobovanie.STAV.M6_Moment_ToleranciaMIN);
//    IF M6_Moment_ToleranciaMIN_REAL > 0 THEN
//        P2_Srobovanie.STAV.M6_Moment_ToleranciaMIN_REAL:= (M6_Moment_ToleranciaMIN_REAL*7.2)/458772;
//    ELSE
//        P2_Srobovanie.STAV.M6_Moment_ToleranciaMIN_REAL:= 0.0;
//    END_IF

    M6_PrevodMomentu.AtlasMinimalnaTolerancia:=P2_Srobovanie.PAR.M6_AtlasCopcoInputs[4];
    P2_Srobovanie.STAV.M6_Moment_ToleranciaMIN_REAL:=M6_PrevodMomentu.ToleranciaMIN;

    (*P2_Srobovanie.STAV.M6_Moment_ToleranciaMIN_REAL:= M6_Moment_ToleranciaMIN_REAL /100;*)

    //Dosiahnutý úhol//
    P2_Srobovanie.STAV.M6_DosiahnutyUhol.0:= P2_Srobovanie.PAR.M6_AtlasCopcoInputs[0].24;
    P2_Srobovanie.STAV.M6_DosiahnutyUhol.1:= P2_Srobovanie.PAR.M6_AtlasCopcoInputs[0].25;
    P2_Srobovanie.STAV.M6_DosiahnutyUhol.2:= P2_Srobovanie.PAR.M6_AtlasCopcoInputs[0].26;
    P2_Srobovanie.STAV.M6_DosiahnutyUhol.3:= P2_Srobovanie.PAR.M6_AtlasCopcoInputs[0].27;
    P2_Srobovanie.STAV.M6_DosiahnutyUhol.4:= P2_Srobovanie.PAR.M6_AtlasCopcoInputs[0].28;
    P2_Srobovanie.STAV.M6_DosiahnutyUhol.5:= P2_Srobovanie.PAR.M6_AtlasCopcoInputs[0].29;
    P2_Srobovanie.STAV.M6_DosiahnutyUhol.6:= P2_Srobovanie.PAR.M6_AtlasCopcoInputs[0].30;
    P2_Srobovanie.STAV.M6_DosiahnutyUhol.7:= P2_Srobovanie.PAR.M6_AtlasCopcoInputs[0].31;
    P2_Srobovanie.STAV.M6_DosiahnutyUhol.8:= P2_Srobovanie.PAR.M6_AtlasCopcoInputs[0].16;
    P2_Srobovanie.STAV.M6_DosiahnutyUhol.9:= P2_Srobovanie.PAR.M6_AtlasCopcoInputs[0].17;
    P2_Srobovanie.STAV.M6_DosiahnutyUhol.10:= P2_Srobovanie.PAR.M6_AtlasCopcoInputs[0].18;
    P2_Srobovanie.STAV.M6_DosiahnutyUhol.11:= P2_Srobovanie.PAR.M6_AtlasCopcoInputs[0].19;
    P2_Srobovanie.STAV.M6_DosiahnutyUhol.12:= P2_Srobovanie.PAR.M6_AtlasCopcoInputs[0].20;
    P2_Srobovanie.STAV.M6_DosiahnutyUhol.13:= P2_Srobovanie.PAR.M6_AtlasCopcoInputs[0].21;
    P2_Srobovanie.STAV.M6_DosiahnutyUhol.14:= P2_Srobovanie.PAR.M6_AtlasCopcoInputs[0].22;
    P2_Srobovanie.STAV.M6_DosiahnutyUhol.15:= P2_Srobovanie.PAR.M6_AtlasCopcoInputs[0].23;

    //Uhol - Tolerancia MAX//
    P2_Srobovanie.STAV.M6_Uhol_ToleranciaMAX.0:= P2_Srobovanie.PAR.M6_AtlasCopcoInputs[2].8;
    P2_Srobovanie.STAV.M6_Uhol_ToleranciaMAX.1:= P2_Srobovanie.PAR.M6_AtlasCopcoInputs[2].9;
    P2_Srobovanie.STAV.M6_Uhol_ToleranciaMAX.2:= P2_Srobovanie.PAR.M6_AtlasCopcoInputs[2].10;
    P2_Srobovanie.STAV.M6_Uhol_ToleranciaMAX.3:= P2_Srobovanie.PAR.M6_AtlasCopcoInputs[2].11;
    P2_Srobovanie.STAV.M6_Uhol_ToleranciaMAX.4:= P2_Srobovanie.PAR.M6_AtlasCopcoInputs[2].12;
    P2_Srobovanie.STAV.M6_Uhol_ToleranciaMAX.5:= P2_Srobovanie.PAR.M6_AtlasCopcoInputs[2].13;
    P2_Srobovanie.STAV.M6_Uhol_ToleranciaMAX.6:= P2_Srobovanie.PAR.M6_AtlasCopcoInputs[2].14;
    P2_Srobovanie.STAV.M6_Uhol_ToleranciaMAX.7:= P2_Srobovanie.PAR.M6_AtlasCopcoInputs[2].15;
    P2_Srobovanie.STAV.M6_Uhol_ToleranciaMAX.8:= P2_Srobovanie.PAR.M6_AtlasCopcoInputs[2].0;
    P2_Srobovanie.STAV.M6_Uhol_ToleranciaMAX.9:= P2_Srobovanie.PAR.M6_AtlasCopcoInputs[2].1;
    P2_Srobovanie.STAV.M6_Uhol_ToleranciaMAX.10:= P2_Srobovanie.PAR.M6_AtlasCopcoInputs[2].2;
    P2_Srobovanie.STAV.M6_Uhol_ToleranciaMAX.11:= P2_Srobovanie.PAR.M6_AtlasCopcoInputs[2].3;
    P2_Srobovanie.STAV.M6_Uhol_ToleranciaMAX.12:= P2_Srobovanie.PAR.M6_AtlasCopcoInputs[2].4;
    P2_Srobovanie.STAV.M6_Uhol_ToleranciaMAX.13:= P2_Srobovanie.PAR.M6_AtlasCopcoInputs[2].5;
    P2_Srobovanie.STAV.M6_Uhol_ToleranciaMAX.14:= P2_Srobovanie.PAR.M6_AtlasCopcoInputs[2].6;
    P2_Srobovanie.STAV.M6_Uhol_ToleranciaMAX.15:= P2_Srobovanie.PAR.M6_AtlasCopcoInputs[2].7;

    //Uhol - Tolerancia MIN//
    P2_Srobovanie.STAV.M6_Uhol_ToleranciaMIN.0:= P2_Srobovanie.PAR.M6_AtlasCopcoInputs[2].24;
    P2_Srobovanie.STAV.M6_Uhol_ToleranciaMIN.1:= P2_Srobovanie.PAR.M6_AtlasCopcoInputs[2].25;
    P2_Srobovanie.STAV.M6_Uhol_ToleranciaMIN.2:= P2_Srobovanie.PAR.M6_AtlasCopcoInputs[2].26;
    P2_Srobovanie.STAV.M6_Uhol_ToleranciaMIN.3:= P2_Srobovanie.PAR.M6_AtlasCopcoInputs[2].27;
    P2_Srobovanie.STAV.M6_Uhol_ToleranciaMIN.4:= P2_Srobovanie.PAR.M6_AtlasCopcoInputs[2].28;
    P2_Srobovanie.STAV.M6_Uhol_ToleranciaMIN.5:= P2_Srobovanie.PAR.M6_AtlasCopcoInputs[2].29;
    P2_Srobovanie.STAV.M6_Uhol_ToleranciaMIN.6:= P2_Srobovanie.PAR.M6_AtlasCopcoInputs[2].30;
    P2_Srobovanie.STAV.M6_Uhol_ToleranciaMIN.7:= P2_Srobovanie.PAR.M6_AtlasCopcoInputs[2].31;
    P2_Srobovanie.STAV.M6_Uhol_ToleranciaMIN.8:= P2_Srobovanie.PAR.M6_AtlasCopcoInputs[2].16;
    P2_Srobovanie.STAV.M6_Uhol_ToleranciaMIN.9:= P2_Srobovanie.PAR.M6_AtlasCopcoInputs[2].17;
    P2_Srobovanie.STAV.M6_Uhol_ToleranciaMIN.10:= P2_Srobovanie.PAR.M6_AtlasCopcoInputs[2].18;
    P2_Srobovanie.STAV.M6_Uhol_ToleranciaMIN.11:= P2_Srobovanie.PAR.M6_AtlasCopcoInputs[2].19;
    P2_Srobovanie.STAV.M6_Uhol_ToleranciaMIN.12:= P2_Srobovanie.PAR.M6_AtlasCopcoInputs[2].20;
    P2_Srobovanie.STAV.M6_Uhol_ToleranciaMIN.13:= P2_Srobovanie.PAR.M6_AtlasCopcoInputs[2].21;
    P2_Srobovanie.STAV.M6_Uhol_ToleranciaMIN.14:= P2_Srobovanie.PAR.M6_AtlasCopcoInputs[2].22;
    P2_Srobovanie.STAV.M6_Uhol_ToleranciaMIN.15:= P2_Srobovanie.PAR.M6_AtlasCopcoInputs[2].23;

END_ACTION
```

#### OvlSkrutkovacichSetov.st
```iecst
ACTION OvlSkrutkovacichSetov:

//***********************************Skrutkovací set M6************************************//
	//Volanie funkcie SequenceControl//
	SequenceControl(SC:= SC_SkrutkovaciSet_M6);

	CASE SC_SkrutkovaciSet_M6.Step OF

		0:
			SC_SkrutkovaciSet_M6.StepName:='0 - Nulovanie';
			P2_Srobovanie.SkrutSet_M6.Cmd.AutomatStart:= FALSE;
			P2_Srobovanie.SkrutSet_M6.Cmd.ManualStartHrniec:= FALSE;
			P2_Srobovanie.SkrutSet_M6.Cmd.PodajSkrutku:= FALSE;
			P2_Srobovanie.CMD.RR_SkrutSetM6_PodajSkrutku:= FALSE;
			P2_Srobovanie.CMD.RR_SkrutSetM6_Zasobnik_RUN:= FALSE;
			P2_Srobovanie.CMD.RR_SkrutSetM6_VysunBrzdu:= FALSE;
			P2_Srobovanie.SkrutSet_M6.Cmd.ManualPresunBrzdu:= FALSE;
			P2_Srobovanie.STAV.SkrutkaM6_READY:= FALSE;
			IF SC_P2_Srobovanie.Step <> 0 THEN
				SC_SkrutkovaciSet_M6.ResetStep:= TRUE;
				SC_SkrutkovaciSet_M6.Step:= 1;
			END_IF

		1:
			SC_SkrutkovaciSet_M6.StepName:='1 - Rozhodnutie o cinnosti';

			IF P2_Srobovanie.Automat THEN
				SC_SkrutkovaciSet_M6.ResetStep:= TRUE;
				SC_SkrutkovaciSet_M6.Step:= 10;
			ELSIF P2_Srobovanie.Manual THEN
				SC_SkrutkovaciSet_M6.ResetStep:= TRUE;
				SC_SkrutkovaciSet_M6.Step:= 20;
			END_IF

		10:
			SC_SkrutkovaciSet_M6.StepName:='10 - Automaticky rezim - cakam na signal podaj skrutku';
			SC_SkrutkovaciSet_M6.IdleTime.PT:= T#2s;
			SC_SkrutkovaciSet_M6.AlarmTime.PT:= T#5s;

			P2_Srobovanie.SkrutSet_M6.Cmd.AutomatStart:= TRUE;

			IF P2_Srobovanie.CMD.PodajSkrutku_M6 THEN
				P2_Srobovanie.CMD.PodajSkrutku_M6:= FALSE;
				SC_SkrutkovaciSet_M6.ResetStep:= TRUE;
				SC_SkrutkovaciSet_M6.Step:= 13;
			END_IF

		13:
			SC_SkrutkovaciSet_M6.StepName:='13 - Automaticky rezim - podanie skrutky do skrutkovacky';
			SC_SkrutkovaciSet_M6.IdleTime.PT:= T#2s;
			SC_SkrutkovaciSet_M6.AlarmTime.PT:= T#5s;

			IF NOT SC_SkrutkovaciSet_M6.Switch1 THEN
				P2_Srobovanie.SkrutSet_M6.Cmd.PodajSkrutku:= TRUE;
				SC_SkrutkovaciSet_M6.Switch1:= TRUE;
			END_IF

			IF P2_Srobovanie.SkrutSet_M6.Status.SkrutkaPripravena THEN
				P2_Srobovanie.STAV.SkrutkaM6_READY:= TRUE;
				P2_Srobovanie.SkrutSet_M6.Cmd.PodajSkrutku:= FALSE;
				SC_SkrutkovaciSet_M6.ResetStep:= TRUE;
				SC_SkrutkovaciSet_M6.Step:= 15;
			ELSIF P2_Srobovanie.SkrutSet_M6.Error.ErrorBit THEN
				P2_Srobovanie.SkrutSet_M6.Cmd.PodajSkrutku:= FALSE;
				P2_Alarmy[239]:= TRUE;
				P2_Pracovisko.STAV.Porucha_ST4:= TRUE;
			END_IF

		15:
			SC_SkrutkovaciSet_M6.StepName:='15 - Automaticky rezim - cakam na zrusenie stavu skrutka M6 READY';
			SC_SkrutkovaciSet_M6.IdleTime.PT:= T#2s;
			SC_SkrutkovaciSet_M6.AlarmTime.PT:= T#5s;

			IF NOT P2_Srobovanie.STAV.SkrutkaM6_READY THEN
				SC_SkrutkovaciSet_M6.ResetStep:= TRUE;
				SC_SkrutkovaciSet_M6.Step:= 10;
			ELSIF P2_Srobovanie.Manual THEN
				P2_Srobovanie.SkrutSet_M6.Cmd.AutomatStart:= FALSE;
				SC_SkrutkovaciSet_M6.ResetStep:= TRUE;
				SC_SkrutkovaciSet_M6.Step:= 20;
			END_IF

		20:
			SC_SkrutkovaciSet_M6.StepName:='20 - Manualny rezim';
			SC_SkrutkovaciSet_M6.IdleTime.PT:= T#2s;
			SC_SkrutkovaciSet_M6.AlarmTime.PT:= T#5s;

			//Ovládanie zásobníka//
			IF P2_Srobovanie.CMD.RR_SkrutSetM6_Zasobnik_RUN THEN
				P2_Srobovanie.SkrutSet_M6.Cmd.AutomatStart:= FALSE;
				P2_Srobovanie.SkrutSet_M6.Cmd.ManualStartHrniec:= TRUE;
			ELSE
				P2_Srobovanie.SkrutSet_M6.Cmd.ManualStartHrniec:= FALSE;
			END_IF

			//Ovládanie brzdy//
			IF P2_Srobovanie.CMD.RR_SkrutSetM6_VysunBrzdu THEN
				P2_Srobovanie.SkrutSet_M6.Cmd.AutomatStart:= FALSE;
				P2_Srobovanie.SkrutSet_M6.Cmd.ManualPresunBrzdu:= TRUE;
			ELSE
				P2_Srobovanie.SkrutSet_M6.Cmd.ManualPresunBrzdu:= FALSE;
			END_IF

			//Podanie skrutky//
			IF P2_Srobovanie.CMD.RR_SkrutSetM6_PodajSkrutku THEN
				P2_Srobovanie.CMD.RR_SkrutSetM6_PodajSkrutku:= FALSE;
				P2_Srobovanie.CMD.RR_SkrutSetM6_Zasobnik_RUN:= FALSE;
				P2_Srobovanie.SkrutSet_M6.Cmd.ManualStartHrniec:= FALSE;
				P2_Srobovanie.SkrutSet_M6.Cmd.ManualPresunBrzdu:= FALSE;
				P2_Srobovanie.CMD.PodajSkrutku_M6:= TRUE;
				SC_SkrutkovaciSet_M6.ResetStep:= TRUE;
				SC_SkrutkovaciSet_M6.Step:= 10;
			END_IF

	END_CASE

	//***********************************Skrutkovací set M4**************************************//
	//Volanie funkcie SequenceControl//
	SequenceControl(SC:= SC_SkrutkovaciSet_M4);

	CASE SC_SkrutkovaciSet_M4.Step OF

		0:
			SC_SkrutkovaciSet_M4.StepName:='0 - Nulovanie';
			P2_Srobovanie.SkrutSet_M4.CMD.ENABLE:= FALSE;
			P2_Srobovanie.SkrutSet_M4.CMD.RucnyRezim:= FALSE;
			P2_Srobovanie.SkrutSet_M4.CMD.PodajSkrutku:= FALSE;
			P2_Srobovanie.SkrutSet_M4.CMD.RR_OtocPodavac_Vstup:= FALSE;
			P2_Srobovanie.SkrutSet_M4.CMD.RR_OtocPodavac_Vystup:= FALSE;
			P2_Srobovanie.SkrutSet_M4.CMD.RR_ZapniVibrolistu:= FALSE;
			P2_Srobovanie.SkrutSet_M4.CMD.RR_ZapniZasobnik:= FALSE;

			IF SC_P2_Srobovanie.Step <> 0 THEN
				SC_SkrutkovaciSet_M4.ResetStep:= TRUE;
				SC_SkrutkovaciSet_M4.Step:= 1;
			END_IF

		1:
			SC_SkrutkovaciSet_M4.StepName:='1 - Rozhodnutie o cinnosti';

			IF P2_Srobovanie.Automat THEN
				SC_SkrutkovaciSet_M4.ResetStep:= TRUE;
				SC_SkrutkovaciSet_M4.Step:= 10;
			ELSIF P2_Srobovanie.Manual THEN
				SC_SkrutkovaciSet_M4.ResetStep:= TRUE;
				SC_SkrutkovaciSet_M4.Step:= 20;
			END_IF

		10:
			SC_SkrutkovaciSet_M4.StepName:='10 - Automaticky rezim - cakam na signal podaj skrutku';
			SC_SkrutkovaciSet_M4.IdleTime.PT:= T#2s;
			SC_SkrutkovaciSet_M4.AlarmTime.PT:= T#5s;

			P2_Srobovanie.SkrutSet_M4.CMD.ENABLE:= TRUE;

			IF P2_Srobovanie.CMD.PodajSkrutku_M4 THEN
				P2_Srobovanie.CMD.PodajSkrutku_M4:= FALSE;
				SC_SkrutkovaciSet_M4.ResetStep:= TRUE;
				SC_SkrutkovaciSet_M4.Step:= 13;
			END_IF

		13:
			SC_SkrutkovaciSet_M4.StepName:='13 - Automaticky rezim - podanie skrutky';
			SC_SkrutkovaciSet_M4.IdleTime.PT:= T#2s;
			SC_SkrutkovaciSet_M4.AlarmTime.PT:= T#5s;

			IF NOT SC_SkrutkovaciSet_M4.Switch1 THEN
				P2_Srobovanie.SkrutSet_M4.CMD.PodajSkrutku:= TRUE;
				SC_SkrutkovaciSet_M4.Switch1:= TRUE;
			END_IF

			IF P2_Srobovanie.SkrutSet_M4.STAV.SkrutkaPripravena THEN
				P2_Srobovanie.SkrutSet_M4.CMD.PodajSkrutku:= FALSE;
				SC_SkrutkovaciSet_M4.ResetStep:= TRUE;
				SC_SkrutkovaciSet_M4.Step:= 15;
			ELSIF P2_Srobovanie.SkrutSet_M4.STAV.ERROR THEN
				P2_Srobovanie.SkrutSet_M4.CMD.PodajSkrutku:= FALSE;
				P2_Alarmy[237]:= TRUE;
				P2_Pracovisko.STAV.Porucha_ST4:= TRUE;
			END_IF

		15:
			SC_SkrutkovaciSet_M4.StepName:='15 - Automaticky rezim - ukoncenie podania skrutkz M4';
			SC_SkrutkovaciSet_M4.IdleTime.PT:= T#2s;
			SC_SkrutkovaciSet_M4.AlarmTime.PT:= T#5s;

			IF P2_Srobovanie.Manual THEN
				SC_SkrutkovaciSet_M4.ResetStep:= TRUE;
				SC_SkrutkovaciSet_M4.Step:= 20;
			ELSE
				SC_SkrutkovaciSet_M4.ResetStep:= TRUE;
				SC_SkrutkovaciSet_M4.Step:= 10;
			END_IF

		20:
			SC_SkrutkovaciSet_M4.StepName:='20 - Manualny rezim';
			SC_SkrutkovaciSet_M4.IdleTime.PT:= T#2s;
			SC_SkrutkovaciSet_M4.AlarmTime.PT:= T#5s;

			P2_Srobovanie.SkrutSet_M4.CMD.ENABLE:= TRUE;
			P2_Srobovanie.SkrutSet_M4.CMD.RucnyRezim:= TRUE;

			//Ovládanie zásobníka//
			IF P2_Srobovanie.CMD.RR_SkrutSetM4_Zasobnik_RUN THEN
				P2_Srobovanie.SkrutSet_M4.CMD.RR_ZapniZasobnik:= TRUE;
			ELSE
				P2_Srobovanie.SkrutSet_M4.CMD.RR_ZapniZasobnik:= FALSE;
			END_IF

			//Ovládanie vibrolišty//
			IF P2_Srobovanie.CMD.RR_SkrutSetM4_Vibrolista_RUN THEN
				P2_Srobovanie.SkrutSet_M4.CMD.RR_ZapniVibrolistu:= TRUE;
			ELSE
				P2_Srobovanie.SkrutSet_M4.CMD.RR_ZapniVibrolistu:= FALSE;
			END_IF

			//Otáčanie podavača skrutiek//
			IF P2_Srobovanie.CMD.RR_SkrutSetM4_OtocPodavac_Vstup THEN
				P2_Srobovanie.SkrutSet_M4.CMD.RR_OtocPodavac_Vstup:= TRUE;
				P2_Srobovanie.CMD.RR_SkrutSetM4_OtocPodavac_Vstup:= FALSE;
			ELSIF P2_Srobovanie.CMD.RR_SkrutSetM4_OtocPodavac_Vystup THEN
				P2_Srobovanie.SkrutSet_M4.CMD.RR_OtocPodavac_Vystup:= TRUE;
				P2_Srobovanie.CMD.RR_SkrutSetM4_OtocPodavac_Vystup:= FALSE;
			END_IF

			//Podanie skrutky//
			IF P2_Srobovanie.CMD.RR_SkrutSetM4_PodajSkrutku THEN
				P2_Srobovanie.CMD.RR_SkrutSetM4_PodajSkrutku:= FALSE;
				P2_Srobovanie.CMD.RR_SkrutSetM4_Zasobnik_RUN:= FALSE;
				P2_Srobovanie.CMD.RR_SkrutSetM4_Vibrolista_RUN:= FALSE;
				P2_Srobovanie.SkrutSet_M4.CMD.RucnyRezim:= TRUE;
				P2_Srobovanie.CMD.PodajSkrutku_M4:= TRUE;
				SC_SkrutkovaciSet_M4.ResetStep:= TRUE;
				SC_SkrutkovaciSet_M4.Step:= 10;
			END_IF

	END_CASE

	//***********************************Skrutkovací set M5***************************************//
	//Volanie funkcie SequenceControl//
	SequenceControl(SC:= SC_SkrutkovaciSet_M5);

	CASE SC_SkrutkovaciSet_M5.Step OF

		0:
			SC_SkrutkovaciSet_M5.StepName:='0 - Nulovanie';
			P2_Srobovanie.SkrutSet_M5.Cmd.AutomatStart:= FALSE;
			P2_Srobovanie.SkrutSet_M5.Cmd.ManualStartHrniec:= FALSE;
			P2_Srobovanie.SkrutSet_M5.Cmd.PodajSkrutku:= FALSE;
			P2_Srobovanie.CMD.RR_SkrutSetM5_PodajSkrutku:= FALSE;
			P2_Srobovanie.CMD.RR_SkrutSetM5_Zasobnik_RUN:= FALSE;
			P2_Srobovanie.CMD.RR_SkrutSetM5_VysunBrzdu:= FALSE;
			P2_Srobovanie.SkrutSet_M5.Cmd.ManualPresunBrzdu:= FALSE;
			P2_Srobovanie.STAV.SkrutkaM5_READY:= FALSE;

			IF SC_P2_Srobovanie.Step <> 0 THEN
				SC_SkrutkovaciSet_M5.ResetStep:= TRUE;
				SC_SkrutkovaciSet_M5.Step:= 1;
			END_IF

		1:
			SC_SkrutkovaciSet_M5.StepName:='1 - Rozhodnutie o cinnosti';

			IF P2_Srobovanie.Automat THEN
				SC_SkrutkovaciSet_M5.ResetStep:= TRUE;
				SC_SkrutkovaciSet_M5.Step:= 10;
			ELSIF P2_Srobovanie.Manual THEN
				SC_SkrutkovaciSet_M5.ResetStep:= TRUE;
				SC_SkrutkovaciSet_M5.Step:= 20;
			END_IF

		10:
			SC_SkrutkovaciSet_M5.StepName:='10 - Automaticky rezim - cakam na signal podaj skrutku';
			SC_SkrutkovaciSet_M5.IdleTime.PT:= T#2s;
			SC_SkrutkovaciSet_M5.AlarmTime.PT:= T#5s;

			P2_Srobovanie.SkrutSet_M5.Cmd.AutomatStart:= TRUE;

			IF P2_Srobovanie.CMD.PodajSkrutku_M5 THEN
				P2_Srobovanie.CMD.PodajSkrutku_M5:= FALSE;
				SC_SkrutkovaciSet_M5.ResetStep:= TRUE;
				SC_SkrutkovaciSet_M5.Step:= 13;
			END_IF

		13:
			SC_SkrutkovaciSet_M5.StepName:='13 - Automaticky rezim - podanie skrutky do skrutkovacky';
			SC_SkrutkovaciSet_M5.IdleTime.PT:= T#2s;
			SC_SkrutkovaciSet_M5.AlarmTime.PT:= T#5s;

			IF NOT SC_SkrutkovaciSet_M5.Switch1 THEN
				P2_Srobovanie.SkrutSet_M5.Cmd.PodajSkrutku:= TRUE;
				SC_SkrutkovaciSet_M5.Switch1:= TRUE;
			END_IF

			IF P2_Srobovanie.SkrutSet_M5.Status.SkrutkaPripravena THEN
				P2_Srobovanie.STAV.SkrutkaM5_READY:= TRUE;
				P2_Srobovanie.SkrutSet_M5.Cmd.PodajSkrutku:= FALSE;
				SC_SkrutkovaciSet_M5.ResetStep:= TRUE;
				SC_SkrutkovaciSet_M5.Step:= 15;
			ELSIF P2_Srobovanie.SkrutSet_M5.Error.ErrorBit THEN
				P2_Srobovanie.SkrutSet_M5.Cmd.PodajSkrutku:= FALSE;
				P2_Alarmy[238]:= TRUE;
				P2_Pracovisko.STAV.Porucha_ST4:= TRUE;
			END_IF

		15:
			SC_SkrutkovaciSet_M5.StepName:='15 - Automaticky rezim - cakam na zrusenie stavu skrutka M5 READY';
			SC_SkrutkovaciSet_M5.IdleTime.PT:= T#2s;
			SC_SkrutkovaciSet_M5.AlarmTime.PT:= T#5s;

			IF NOT P2_Srobovanie.STAV.SkrutkaM5_READY THEN
				SC_SkrutkovaciSet_M5.ResetStep:= TRUE;
				SC_SkrutkovaciSet_M5.Step:= 10;
			ELSIF P2_Srobovanie.Manual THEN
				P2_Srobovanie.SkrutSet_M5.Cmd.AutomatStart:= FALSE;
				SC_SkrutkovaciSet_M5.ResetStep:= TRUE;
				SC_SkrutkovaciSet_M5.Step:= 20;
			END_IF

		20:
			SC_SkrutkovaciSet_M5.StepName:='20 - Manualny rezim';
			SC_SkrutkovaciSet_M5.IdleTime.PT:= T#2s;
			SC_SkrutkovaciSet_M5.AlarmTime.PT:= T#5s;

			//Ovládanie zásobníka//
			IF P2_Srobovanie.CMD.RR_SkrutSetM5_Zasobnik_RUN THEN
				P2_Srobovanie.SkrutSet_M5.Cmd.AutomatStart:= FALSE;
				P2_Srobovanie.SkrutSet_M5.Cmd.ManualStartHrniec:= TRUE;
			ELSE
				P2_Srobovanie.SkrutSet_M5.Cmd.ManualStartHrniec:= FALSE;
			END_IF

			//Ovládanie brzdy//
			IF P2_Srobovanie.CMD.RR_SkrutSetM5_VysunBrzdu THEN
				P2_Srobovanie.SkrutSet_M5.Cmd.AutomatStart:= FALSE;
				P2_Srobovanie.SkrutSet_M5.Cmd.ManualPresunBrzdu:= TRUE;
			ELSE
				P2_Srobovanie.SkrutSet_M5.Cmd.ManualPresunBrzdu:= FALSE;
			END_IF

			//Podanie skrutky//
			IF P2_Srobovanie.CMD.RR_SkrutSetM5_PodajSkrutku THEN
				P2_Srobovanie.CMD.RR_SkrutSetM5_PodajSkrutku:= FALSE;
				P2_Srobovanie.CMD.RR_SkrutSetM5_Zasobnik_RUN:= FALSE;
				P2_Srobovanie.SkrutSet_M5.Cmd.ManualStartHrniec:= FALSE;
				P2_Srobovanie.SkrutSet_M5.Cmd.ManualPresunBrzdu:= FALSE;
				P2_Srobovanie.CMD.PodajSkrutku_M5:= TRUE;
				SC_SkrutkovaciSet_M5.ResetStep:= TRUE;
				SC_SkrutkovaciSet_M5.Step:= 10;
			END_IF

	END_CASE

END_ACTION
```

### Program Logical/Program/Pracovisko_2/P2_Robot (IEC)

#### Main.st - Init, cyclic, exit code
```iecst
PROGRAM _INIT
	(* Insert code here *)

END_PROGRAM

PROGRAM _CYCLIC

	//Volanie funkcie SequenceControl//
	SequenceControl(SC:= SC_P2_Robot);

	//Volanie podprogramov//
	ProfinetKomunikaciaRobot;

	//Reset sekcie //
	IF P2_Robot.Reset THEN
		SC_P2_Robot.Step:= 0;
		P2_Robot.Reset:= FALSE;
	ELSIF NOT Safety.STAV.Linka_ZonaCS_AKTIVNA THEN
		SC_P2_Robot.Step:= 0;
	END_IF

	CASE SC_P2_Robot.Step OF

		0:
			SC_P2_Robot.StepName:='0 - Nulovanie';
			P2_Robot.Automat:= FALSE;
			P2_Robot.KoniecCyklu:= FALSE;
			P2_Robot.Manual:= FALSE;
			P2_Robot.Reset:= FALSE;
			P2_Robot.STAV.PoINIT:= FALSE;
			P2_Robot.COM_OUT.Odparkovanie:= FALSE;
			P2_Robot.COM_OUT.PP_na_Main:= FALSE;
			P2_Robot.COM_OUT.Reset_CS:= FALSE;
			P2_Robot.COM_OUT.StartProgramu:= FALSE;
			P2_Robot.COM_OUT.StartProgramuMain:= FALSE;
			P2_Robot.COM_OUT.VypniMotory:= FALSE;
			P2_Robot.COM_OUT.ZapniMotory:= FALSE;
			IF P2_Robot.COM_IN.Stav_RezimAUTOMAT AND P2_Robot.COM_IN.Stav_ProgramRUN THEN
				P2_Robot.COM_OUT.StopProgramu:= TRUE;
			ELSE
				P2_Robot.COM_OUT.StopProgramu:= FALSE;
			END_IF
			IF Safety.STAV.Linka_ZonaCS_AKTIVNA AND
				P2_Pracovisko.STAV.HardwareBunky_OK AND
				NOT P2_Pracovisko.STAV.Porucha_ST2 AND
				NOT P2_Pracovisko.STAV.Porucha_ST3 AND
				NOT P2_Pracovisko.STAV.Porucha_ST4 AND
				NOT P2_Pracovisko.STAV.Porucha_ST5 AND
				NOT P2_Robot.COM_IN.Stav_ProgramRUN THEN
				P2_Robot.COM_OUT.StopProgramu:= FALSE;
				SC_P2_Robot.ResetStep:= TRUE;
				SC_P2_Robot.Step:= 1;
			END_IF

		1:
			SC_P2_Robot.StepName:='1 - Cakam na spustenie vyroby';
			P2_Robot.KoniecCyklu:= FALSE;
			IF P2_Robot.Automat THEN
				SC_P2_Robot.Step:= 2;
			ELSIF P2_Robot.Manual THEN
				SC_P2_Robot.Step:= 700;
			END_IF

			//********************************************************Inicializácia****************************************************************************//

		2:
			SC_P2_Robot.StepName:='2 - Inicializacia - cakam na spustenie inicializacie';
			SC_P2_Robot.IdleTime.PT:= T#500ms;
			SC_P2_Robot.AlarmTime.PT:= T#5s;

			SC_P2_Robot.IdleTime.IN:= TRUE;

			P2_Robot.COM_OUT.VypniMotory:= TRUE;

			IF SC_P2_Robot.IdleTime.Q AND P2_Cistenie.STAV.PoINIT THEN
				SC_P2_Robot.ResetStep:= TRUE;
				SC_P2_Robot.Step:= 3;
			END_IF

		3:
			SC_P2_Robot.StepName:='2 - Inicializacia - kontrolujem central stop robota';
			SC_P2_Robot.IdleTime.PT:= T#500ms;
			SC_P2_Robot.AlarmTime.PT:= T#5s;

			IF P2_Robot.COM_IN.Stav_RobotCS THEN
				P2_Robot.COM_OUT.Reset_CS:= TRUE;
			END_IF

			IF NOT P2_Robot.COM_IN.Stav_RobotCS THEN
				P2_Robot.COM_OUT.Reset_CS:= FALSE;
				SC_P2_Robot.ResetStep:= TRUE;
				SC_P2_Robot.Step:= 4;
			END_IF

		4:
			SC_P2_Robot.StepName:='4 - Inicializacia - zapinam motory robota';
			SC_P2_Robot.IdleTime.PT:= T#3s;
			SC_P2_Robot.AlarmTime.PT:= T#5s;
			SC_P2_Robot.IdleTime.IN:= TRUE;

			IF NOT P2_Robot.COM_IN.Stav_MotoryON THEN
				P2_Robot.COM_OUT.VypniMotory:= FALSE;
				P2_Robot.COM_OUT.ZapniMotory:= TRUE;
				SC_P2_Robot.IdleTime.IN:= TRUE;
			END_IF

			IF P2_Robot.COM_IN.Stav_MotoryON THEN
				P2_Robot.COM_OUT.ZapniMotory:= FALSE;
				SC_P2_Robot.ResetStep:= TRUE;
				SC_P2_Robot.Step:= 6;
			END_IF

		6:
			SC_P2_Robot.StepName:='6 - Inicializacia - spustam program robota od zaciatku';
			SC_P2_Robot.IdleTime.PT:= T#2s;
			SC_P2_Robot.AlarmTime.PT:= T#10s;

			SC_P2_Robot.IdleTime.IN:= P2_Robot.COM_IN.Stav_ProgramRUN;

			IF NOT SC_P2_Robot.Switch1 THEN
				P2_Robot.COM_OUT.StartProgramuMain:= TRUE;
				SC_P2_Robot.AlarmTime.IN:= TRUE;
				SC_P2_Robot.Switch1:= TRUE;
			END_IF

			IF SC_P2_Robot.IdleTime.Q AND P2_Robot.COM_IN.Stav_VystupyZresetovane THEN
				P2_Robot.COM_OUT.StartProgramuMain:= FALSE;
				P2_Robot.STAV.PoINIT:= TRUE;
				SC_P2_Robot.ResetStep:= TRUE;
				SC_P2_Robot.Step:= 100;
			ELSIF SC_P2_Robot.AlarmTime.Q THEN
				SC_P2_Robot.ResetStep:= TRUE;
				SC_P2_Robot.Step:= 0;
			END_IF

			//********************************************************Automatický režim****************************************************************************//

		100:
			SC_P2_Robot.StepName:='100 - Automaticky Rezim - cakam na ukoncenie programu robota';
			SC_P2_Robot.IdleTime.PT:= T#200ms;
			SC_P2_Robot.AlarmTime.PT:= T#5s;

			IF P2_Robot.KoniecCyklu AND NOT P2_StoperSrobovania.Automat AND NOT P2_StoperZvarania.Automat AND P2_Robot.COM_IN.Stav_RobotOdparkovany THEN
				SC_P2_Robot.ResetStep:= TRUE;
				SC_P2_Robot.Step:= 0;
			ELSIF NOT P2_Robot.COM_IN.Stav_ProgramRUN THEN
				SC_P2_Robot.ResetStep:= TRUE;
				SC_P2_Robot.Step:= 0;
			END_IF

			//*******************************************************Manuálny režim*******************************************************************************//

		700:
			SC_P2_Robot.StepName:='700 - Manualny Rezim';
			SC_P2_Robot.IdleTime.PT:= T#8s;
			SC_P2_Robot.AlarmTime.PT:= T#5s;

	END_CASE

	//Zrušenie signálu výmena gripra 4F5F//
	IF P2_Robot.COM_OUT.ZmenaGripra_4F5F AND P2_Robot.COM_IN.Stav_Griper4F5F_Vymeneny THEN
		P2_Robot.COM_OUT.ZmenaGripra_4F5F:= FALSE;
	END_IF

	//Zrušenie signálu výmena gripra 5H//
	IF P2_Robot.COM_OUT.ZmenaGripra_5H AND P2_Robot.COM_IN.Stav_Griper5H_Vymeneny THEN
		P2_Robot.COM_OUT.ZmenaGripra_5H:= FALSE;
	END_IF

	//Zrušenie signálu výmena gripra čistenia Power CP//
	IF P2_Robot.COM_OUT.ZmenaGripra_Cistenie AND P2_Robot.COM_IN.Stav_GriperCistenia_Vymeneny THEN
		P2_Robot.COM_OUT.ZmenaGripra_Cistenie:= FALSE;
	END_IF

END_PROGRAM

PROGRAM _EXIT
	(* Insert code here *)

END_PROGRAM
```

#### ProfinetKomunikaciaRobot.st
```iecst
ACTION ProfinetKomunikaciaRobot:

	//Vstupy z Robota do PLC//
	P2_Robot.COM_IN.Stav_RezimAUTOMAT:= P2_Robot.COM_IN.BYTE_IN[0].0;
	P2_Robot.COM_IN.Stav_ProgramRUN:= P2_Robot.COM_IN.BYTE_IN[0].1;
	P2_Robot.COM_IN.Stav_MotoryOFF:= P2_Robot.COM_IN.BYTE_IN[0].2;
	P2_Robot.COM_IN.Stav_MotoryON:= P2_Robot.COM_IN.BYTE_IN[0].3;
	P2_Robot.COM_IN.Stav_RobotCS:= P2_Robot.COM_IN.BYTE_IN[0].4;
	P2_Robot.COM_IN.BYTE_IN[0].5;
	P2_Robot.COM_IN.BYTE_IN[0].6;
	P2_Robot.COM_IN.BYTE_IN[0].7;

	P2_Robot.OUT.Griper_ZATVOR:= P2_Robot.COM_IN.BYTE_IN[1].0;
	P2_Robot.OUT.Griper_OTVOR:= P2_Robot.COM_IN.BYTE_IN[1].1;
	P2_Robot.OUT.ZaistiGriper:= P2_Robot.COM_IN.BYTE_IN[1].2;
	P2_Robot.OUT.OdistiGriper:= P2_Robot.COM_IN.BYTE_IN[1].3;
	P2_Robot.OUT.Model5H_Vakum_ON:= P2_Robot.COM_IN.BYTE_IN[1].4;
	P2_Robot.OUT.Model45F_Vakum_ON:= P2_Robot.COM_IN.BYTE_IN[1].5;
	P2_Robot.COM_IN.Stav_Busbary5H_Odobrate:= P2_Robot.COM_IN.BYTE_IN[1].6;
	P2_Robot.COM_IN.Stav_Busbary5F_Odobrate:= P2_Robot.COM_IN.BYTE_IN[1].7;

	P2_Robot.COM_IN.Stav_Busbary4F_Odobrate:= P2_Robot.COM_IN.BYTE_IN[2].0;
	P2_Robot.COM_IN.Stav_Busbary5H_Polozene:= P2_Robot.COM_IN.BYTE_IN[2].1;
	P2_Robot.COM_IN.Stav_Busbary5F_Polozene:= P2_Robot.COM_IN.BYTE_IN[2].2;
	P2_Robot.COM_IN.Stav_Busbary4F_Polozene:= P2_Robot.COM_IN.BYTE_IN[2].3;
	P2_Robot.COM_IN.Stav_RobotPoziciaCakania:= P2_Robot.COM_IN.BYTE_IN[2].4;
	P2_Robot.COM_IN.Stav_Filter5H_Dotlaceny:= P2_Robot.COM_IN.BYTE_IN[2].5;
	P2_Robot.COM_IN.BYTE_IN[2].6;
	P2_Robot.COM_IN.Stav_Cistenie_PowerCP_Odobrate:= P2_Robot.COM_IN.BYTE_IN[2].7;

	P2_Robot.COM_IN.BYTE_IN[3].0;
	P2_Robot.COM_IN.BYTE_IN[3].1;
	P2_Robot.COM_IN.Stav_Cistenie_Otacanie_Ukoncene:= P2_Robot.COM_IN.BYTE_IN[3].2;
	P2_Robot.COM_IN.Stav_Cistenie_PowerCP_v_Cisteni:= P2_Robot.COM_IN.BYTE_IN[3].3;
	P2_Robot.COM_IN.Stav_Cistenie_PowerCP_Polozene:= P2_Robot.COM_IN.BYTE_IN[3].4;
	P2_Robot.COM_IN.BYTE_IN[3].5;
	P2_Robot.COM_IN.BYTE_IN[3].6;
	P2_Robot.COM_IN.Stav_LavyMvCase5H_Odobraty:= P2_Robot.COM_IN.BYTE_IN[3].7;

	P2_Robot.COM_IN.Stav_LavyMvCase5F_Odobraty:= P2_Robot.COM_IN.BYTE_IN[4].0;
	P2_Robot.COM_IN.Stav_LavyMvCase4F_Odobraty:= P2_Robot.COM_IN.BYTE_IN[4].1;
	P2_Robot.COM_IN.Stav_PravyMvCase5H_Odobraty:= P2_Robot.COM_IN.BYTE_IN[4].2;
	P2_Robot.COM_IN.Stav_PravyMvCase5F_Odobraty:= P2_Robot.COM_IN.BYTE_IN[4].3;
	P2_Robot.COM_IN.Stav_PravyMvCase4F_Odobraty:= P2_Robot.COM_IN.BYTE_IN[4].4;
	P2_Robot.COM_IN.Stav_TopCover5H_Odobraty:= P2_Robot.COM_IN.BYTE_IN[4].5;
	P2_Robot.COM_IN.Stav_TopCover5F_Odobraty:= P2_Robot.COM_IN.BYTE_IN[4].6;
	P2_Robot.COM_IN.Stav_TopCover4F_Odobraty:= P2_Robot.COM_IN.BYTE_IN[4].7;

	P2_Robot.OUT.Model5H_Vakum_OFF:= P2_Robot.COM_IN.BYTE_IN[5].0;
	P2_Robot.OUT.Model45F_Vakum_OFF:= P2_Robot.COM_IN.BYTE_IN[5].1;
	P2_Robot.OUT.PneuZamokUchopovaca_ODOMKNI:= P2_Robot.COM_IN.BYTE_IN[5].2;
	P2_Robot.COM_IN.Stav_LavyMvCase5H_Polozeny:= P2_Robot.COM_IN.BYTE_IN[5].3;
	P2_Robot.COM_IN.Stav_LavyMvCase5F_Polozeny:= P2_Robot.COM_IN.BYTE_IN[5].4;
	P2_Robot.COM_IN.Stav_LavyMvCase4F_Polozeny:= P2_Robot.COM_IN.BYTE_IN[5].5;
	P2_Robot.COM_IN.Stav_PravyMvCase5H_Polozeny:= P2_Robot.COM_IN.BYTE_IN[5].6;
	P2_Robot.COM_IN.Stav_PravyMvCase5F_Polozeny:= P2_Robot.COM_IN.BYTE_IN[5].7;

	P2_Robot.COM_IN.Stav_PravyMvCase4F_Polozeny:= P2_Robot.COM_IN.BYTE_IN[6].0;
	P2_Robot.COM_IN.Stav_TopCover5H_Polozeny:= P2_Robot.COM_IN.BYTE_IN[6].1;
	P2_Robot.COM_IN.Stav_TopCover5F_Polozeny:= P2_Robot.COM_IN.BYTE_IN[6].2;
	P2_Robot.COM_IN.Stav_TopCover4F_Polozeny:= P2_Robot.COM_IN.BYTE_IN[6].3;
	P2_Robot.COM_IN.Stav_RobotOdparkovany:= P2_Robot.COM_IN.BYTE_IN[6].4;
	P2_Robot.COM_IN.Stav_RobotBezpPozicia_Srobovanie:= P2_Robot.COM_IN.BYTE_IN[6].5;
	P2_Robot.COM_IN.Stav_RobotBezpPozicia_Zvaranie:= P2_Robot.COM_IN.BYTE_IN[6].6;
	P2_Robot.COM_IN.Stav_VystupyZresetovane:= P2_Robot.COM_IN.BYTE_IN[6].7;

	P2_Robot.COM_IN.Stav_BusbaryUvolnene:= P2_Robot.COM_IN.BYTE_IN[7].0;
    P2_Robot.COM_IN.Stav_Griper4F5F_Vymeneny:= P2_Robot.COM_IN.BYTE_IN[7].1;
    P2_Robot.COM_IN.Stav_Griper5H_Vymeneny:= P2_Robot.COM_IN.BYTE_IN[7].2;
    P2_Robot.COM_IN.Stav_GriperCistenia_Vymeneny:= P2_Robot.COM_IN.BYTE_IN[7].3;
	P2_Robot.COM_IN.Stav_RobotOdoberaCover:= P2_Robot.COM_IN.BYTE_IN[7].4;

	//Vystupy z PLC do Robota//
	P2_Robot.COM_OUT.BYTE_OUT[0].0:= P2_Robot.COM_OUT.VypniMotory;
	P2_Robot.COM_OUT.BYTE_OUT[0].1:= P2_Robot.COM_OUT.ZapniMotory;
	P2_Robot.COM_OUT.BYTE_OUT[0].2:= P2_Robot.COM_OUT.PP_na_Main;
	P2_Robot.COM_OUT.BYTE_OUT[0].3:= P2_Robot.COM_OUT.StartProgramu;
	P2_Robot.COM_OUT.BYTE_OUT[0].4:= P2_Robot.COM_OUT.StartProgramuMain;
	P2_Robot.COM_OUT.BYTE_OUT[0].5:= P2_Robot.COM_OUT.StopProgramu;
	P2_Robot.COM_OUT.BYTE_OUT[0].6:= P2_Robot.COM_OUT.Reset_CS;
	P2_Robot.COM_OUT.BYTE_OUT[0].7;

	P2_Robot.COM_OUT.BYTE_OUT[1].0:= P2_Robot.IN.TypGripra_5H;
	P2_Robot.COM_OUT.BYTE_OUT[1].1:= P2_Robot.IN.TypGripra_45F;
	P2_Robot.COM_OUT.BYTE_OUT[1].2:= P2_Robot.IN.TypGripra_MvCase;
	P2_Robot.COM_OUT.BYTE_OUT[1].3:= P2_Robot.IN.Griper45F_Otvoreny;
	P2_Robot.COM_OUT.BYTE_OUT[1].4:= P2_Robot.IN.Griper45F_DrziBusbary;
	P2_Robot.COM_OUT.BYTE_OUT[1].5:= P2_Robot.IN.Griper45F_Zatvoreny;
	P2_Robot.COM_OUT.BYTE_OUT[1].6:= P2_Robot.IN.Griper5H_Otvoreny;
	P2_Robot.COM_OUT.BYTE_OUT[1].7:= P2_Robot.IN.Griper5H_DrziBusbary;

	P2_Robot.COM_OUT.BYTE_OUT[2].0:= P2_Robot.IN.Griper5H_Zatvoreny;
	P2_Robot.COM_OUT.BYTE_OUT[2].1:= P2_Robot.IN.GriperMvCase_Otvoreny;
	P2_Robot.COM_OUT.BYTE_OUT[2].2:= P2_Robot.IN.GriperMvCase_DrziMvCase;
	P2_Robot.COM_OUT.BYTE_OUT[2].3:= P2_Robot.IN.GriperMvCase_DrziPowerCP;
	P2_Robot.COM_OUT.BYTE_OUT[2].4:= P2_Robot.IN.GriperMvCase_Zatvoreny;
	P2_Robot.COM_OUT.BYTE_OUT[2].5:= P2_Robot.IN.Model5H_Vakum_OK;
	P2_Robot.COM_OUT.BYTE_OUT[2].6:= P2_Robot.IN.Model45F_Vakum_OK;
	P2_Robot.COM_OUT.BYTE_OUT[2].7:= P2_Robot.COM_OUT.Odober_Busbary5H;

	P2_Robot.COM_OUT.BYTE_OUT[3].0:= P2_Robot.COM_OUT.Odober_Busbary5F;
	P2_Robot.COM_OUT.BYTE_OUT[3].1:= P2_Robot.COM_OUT.Odober_Busbary4F;
	P2_Robot.COM_OUT.BYTE_OUT[3].2:= P2_Robot.COM_OUT.Poloz_Busbary5H;
	P2_Robot.COM_OUT.BYTE_OUT[3].3:= P2_Robot.COM_OUT.Poloz_Busbary5F;
	P2_Robot.COM_OUT.BYTE_OUT[3].4:= P2_Robot.COM_OUT.Poloz_Busbary4F;
	P2_Robot.COM_OUT.BYTE_OUT[3].5:= P2_Robot.COM_OUT.Presun_CakaciaPozicia;
	P2_Robot.COM_OUT.BYTE_OUT[3].6:= P2_Robot.COM_OUT.Dotlac_Filter5H;
	P2_Robot.COM_OUT.BYTE_OUT[3].7;

	P2_Robot.COM_OUT.BYTE_OUT[4].0:= P2_Robot.COM_OUT.Cistenie_OdoberPowerCP_5H;
	P2_Robot.COM_OUT.BYTE_OUT[4].1:= P2_Robot.COM_OUT.Cistenie_OdoberPowerCP_5F;
	P2_Robot.COM_OUT.BYTE_OUT[4].2:= P2_Robot.COM_OUT.Cistenie_OdoberPowerCP_4F;
	P2_Robot.COM_OUT.BYTE_OUT[4].3;
	P2_Robot.COM_OUT.BYTE_OUT[4].4;
	P2_Robot.COM_OUT.BYTE_OUT[4].5;
	P2_Robot.COM_OUT.BYTE_OUT[4].6:= P2_Robot.COM_OUT.Cistenie_PolozPowerCP_5H;
	P2_Robot.COM_OUT.BYTE_OUT[4].7:= P2_Robot.COM_OUT.Cistenie_PolozPowerCP_5F;

	P2_Robot.COM_OUT.BYTE_OUT[5].0:= P2_Robot.COM_OUT.Cistenie_PolozPowerCP_4F;
	P2_Robot.COM_OUT.BYTE_OUT[5].1:= P2_Robot.COM_OUT.Odober_LavyMvCase5H;
	P2_Robot.COM_OUT.BYTE_OUT[5].2:= P2_Robot.COM_OUT.Odober_LavyMvCase5F;
	P2_Robot.COM_OUT.BYTE_OUT[5].3:= P2_Robot.COM_OUT.Odober_LavyMvCase4F;
	P2_Robot.COM_OUT.BYTE_OUT[5].4:= P2_Robot.COM_OUT.Odober_PravyMvCase5H;
	P2_Robot.COM_OUT.BYTE_OUT[5].5:= P2_Robot.COM_OUT.Odober_PravyMvCase5F;
	P2_Robot.COM_OUT.BYTE_OUT[5].6:= P2_Robot.COM_OUT.Odober_PravyMvCase4F;
	P2_Robot.COM_OUT.BYTE_OUT[5].7:= P2_Robot.COM_OUT.Odober_TopCover5H;

	P2_Robot.COM_OUT.BYTE_OUT[6].0:= P2_Robot.COM_OUT.Odober_TopCover5F;
	P2_Robot.COM_OUT.BYTE_OUT[6].1:= P2_Robot.COM_OUT.Odober_TopCover4F;
	P2_Robot.COM_OUT.BYTE_OUT[6].2:= P2_Robot.IN.DokStanica_PritomGripraBusbar5H;
	P2_Robot.COM_OUT.BYTE_OUT[6].3:= P2_Robot.IN.DokStanica_PritomGripraBusbar45F;
	P2_Robot.COM_OUT.BYTE_OUT[6].4:= P2_Robot.IN.DokStanica_PritomGripraMvCase;
	P2_Robot.COM_OUT.BYTE_OUT[6].5:= P2_Robot.COM_OUT.Cistenie_BezpecnaPozicia;
	P2_Robot.COM_OUT.BYTE_OUT[6].6:= P2_Robot.COM_OUT.Cistenie_OtacajPowerCP;
	P2_Robot.COM_OUT.BYTE_OUT[6].7:= P2_Robot.COM_OUT.ManipSrobovania_BezpecnaPozicia;

	P2_Robot.COM_OUT.BYTE_OUT[7].0:= P2_Robot.COM_OUT.Poloz_LavyMvCase5H;
	P2_Robot.COM_OUT.BYTE_OUT[7].1:= P2_Robot.COM_OUT.Poloz_LavyMvCase5F;
	P2_Robot.COM_OUT.BYTE_OUT[7].2:= P2_Robot.COM_OUT.Poloz_LavyMvCase4F;
	P2_Robot.COM_OUT.BYTE_OUT[7].3:= P2_Robot.COM_OUT.Poloz_PravyMvCase5H;
	P2_Robot.COM_OUT.BYTE_OUT[7].4:= P2_Robot.COM_OUT.Poloz_PravyMvCase5F;
	P2_Robot.COM_OUT.BYTE_OUT[7].5:= P2_Robot.COM_OUT.Poloz_PravyMvCase4F;
	P2_Robot.COM_OUT.BYTE_OUT[7].6:= P2_Robot.COM_OUT.Poloz_TopCover5H;
	P2_Robot.COM_OUT.BYTE_OUT[7].7:= P2_Robot.COM_OUT.Poloz_TopCover5F;

	P2_Robot.COM_OUT.BYTE_OUT[8].0:= P2_Robot.COM_OUT.Poloz_TopCover4F;
	P2_Robot.COM_OUT.BYTE_OUT[8].1:= P2_Robot.COM_OUT.Odparkovanie;
	P2_Robot.COM_OUT.BYTE_OUT[8].2:= P2_Robot.COM_OUT.Zvaranie_BezpecnaPozicia;
	P2_Robot.COM_OUT.BYTE_OUT[8].3:= P2_Robot.COM_OUT.UvolniBusbary;
    P2_Robot.COM_OUT.BYTE_OUT[8].4:= P2_Robot.COM_OUT.ZmenaGripra_4F5F;
    P2_Robot.COM_OUT.BYTE_OUT[8].5:= P2_Robot.COM_OUT.ZmenaGripra_5H;
    P2_Robot.COM_OUT.BYTE_OUT[8].6:= P2_Robot.COM_OUT.ZmenaGripra_Cistenie;
    P2_Robot.COM_OUT.BYTE_OUT[8].7:= P2_Robot.COM_OUT.ZopakujOdoberanie;

END_ACTION
```

### Program Logical/Program/Pracovisko_2/P2_StoperZvarania (IEC)
